  A_360_01_SQ5_A405_OPT_EKSKL : FbBinaryValue_Medium (2004) := (                _sDescription := 'Optimizer',                 _sActiveText := 'Utkoblet',                 _sInactiveText := 'Innkoblet'           );
  A_360_01_SQ5_A405_A1 : FbBinaryInput_Large (2008) := (                _sDescription := 'Luftmengde Sjeld',                 _sActiveText := 'Feil på luftmengde',                 _sInactiveText := 'Ingen feil',                 _udiNotificationClass := 22           );
  A_360_01_SQ5_A405_A2 : FbBinaryInput_Large (2009) := (                _sDescription := 'Kommunikasjonovervåking',                 _sActiveText := 'Kommunikasjonsfeil',                 _sInactiveText := 'Ingen feil',                 _udiNotificationClass := 22           );
  A_360_01_SQ4_A401_2_VOL : FbAnalogInput_Medium (2010) := (                _sDescription := 'Faktisk luftmengde',                 _rCov_Increment := 1,                 _eUnits := WagoTypesBacnet.eBACnetUnits.UNIT_CUBIC_METERS_PER_HOUR           );
  A_360_01_SQ4_A401_2_SP : FbAnalogValue_Medium (2015) := (                _sDescription := 'Settpunkt',                 _rCov_Increment := 1,                 _eUnits := WagoTypesBacnet.eBACnetUnits.UNIT_CUBIC_METERS_PER_HOUR           );
  A_360_01_SQ4_A401_2_VMIN : FbAnalogValue_Medium (2016) := (                _sDescription := 'Minste luftmengde',                 _rCov_Increment := 1,                 _eUnits := WagoTypesBacnet.eBACnetUnits.UNIT_CUBIC_METERS_PER_HOUR           );
  A_360_01_SQ4_A401_2_VMAX : FbAnalogValue_Medium (2017) := (                _sDescription := 'Største luftmengde',                 _rCov_Increment := 1,                 _eUnits := WagoTypesBacnet.eBACnetUnits.UNIT_CUBIC_METERS_PER_HOUR           );
  A_360_01_SQ4_A401_2_FB : FbAnalogInput_Medium (2011) := (                _sDescription := 'Spjeldvinkel',                 _rCov_Increment := 1,                 _eUnits := WagoTypesBacnet.eBACnetUnits.UNIT_PERCENT           );
  A_360_01_SQ4_A401_2_C : FbAnalogOutput_Medium (2005) := (                _sDescription := 'Pådrag',                 _rCov_Increment := 1,                 _eUnits := WagoTypesBacnet.eBACnetUnits.UNIT_PERCENT           );
  A_360_01_SQ4_A401_2_KMD : FbMultiStateValue_Large (2005) := (                _sDescription := 'Manuell overstyring',                 _udiNumberOfStates := 8           );
  A_360_01_SQ4_A401_2_OPT_EKSKL : FbBinaryValue_Medium (2005) := (                _sDescription := 'Optimizer',                 _sActiveText := 'Utkoblet',                 _sInactiveText := 'Innkoblet'           );
  A_360_01_SQ4_A401_2_A1 : FbBinaryInput_Large (2010) := (                _sDescription := 'Luftmengde Sjeld',                 _sActiveText := 'Feil på luftmengde',                 _sInactiveText := 'Ingen feil',                 _udiNotificationClass := 22           );
  A_360_01_SQ4_A401_2_A2 : FbBinaryInput_Large (2011) := (                _sDescription := 'Kommunikasjonovervåking',                 _sActiveText := 'Kommunikasjonsfeil',                 _sInactiveText := 'Ingen feil',                 _udiNotificationClass := 22           );
  A_360_01_SQ4_A401_1_VOL : FbAnalogInput_Medium (2012) := (                _sDescription := 'Faktisk luftmengde',                 _rCov_Increment := 1,                 _eUnits := WagoTypesBacnet.eBACnetUnits.UNIT_CUBIC_METERS_PER_HOUR           );
  A_360_01_SQ4_A401_1_SP : FbAnalogValue_Medium (2018) := (                _sDescription := 'Settpunkt',                 _rCov_Increment := 1,                 _eUnits := WagoTypesBacnet.eBACnetUnits.UNIT_CUBIC_METERS_PER_HOUR           );
  A_360_01_SQ4_A401_1_VMIN : FbAnalogValue_Medium (2019) := (                _sDescription := 'Minste luftmengde',                 _rCov_Increment := 1,                 _eUnits := WagoTypesBacnet.eBACnetUnits.UNIT_CUBIC_METERS_PER_HOUR           );
  A_360_01_SQ4_A401_1_VMAX : FbAnalogValue_Medium (2020) := (                _sDescription := 'Største luftmengde',                 _rCov_Increment := 1,                 _eUnits := WagoTypesBacnet.eBACnetUnits.UNIT_CUBIC_METERS_PER_HOUR           );
  A_360_01_SQ4_A401_1_FB : FbAnalogInput_Medium (2013) := (                _sDescription := 'Spjeldvinkel',                 _rCov_Increment := 1,                 _eUnits := WagoTypesBacnet.eBACnetUnits.UNIT_PERCENT           );
  A_360_01_SQ4_A401_1_C : FbAnalogOutput_Medium (2006) := (                _sDescription := 'Pådrag',                 _rCov_Increment := 1,                 _eUnits := WagoTypesBacnet.eBACnetUnits.UNIT_PERCENT           );
  A_360_01_SQ4_A401_1_KMD : FbMultiStateValue_Large (2006) := (                _sDescription := 'Manuell overstyring',                 _udiNumberOfStates := 8           );
  A_360_01_SQ4_A401_1_OPT_EKSKL : FbBinaryValue_Medium (2006) := (                _sDescription := 'Optimizer',                 _sActiveText := 'Utkoblet',                 _sInactiveText := 'Innkoblet'           );
  A_360_01_SQ4_A401_1_A1 : FbBinaryInput_Large (2012) := (                _sDescription := 'Luftmengde Sjeld',                 _sActiveText := 'Feil på luftmengde',                 _sInactiveText := 'Ingen feil',                 _udiNotificationClass := 22           );
  A_360_01_SQ4_A401_1_A2 : FbBinaryInput_Large (2013) := (                _sDescription := 'Kommunikasjonovervåking',                 _sActiveText := 'Kommunikasjonsfeil',                 _sInactiveText := 'Ingen feil',                 _udiNotificationClass := 22           );
  A_360_01_SQ4_A401_VOL : FbAnalogInput_Medium (2014) := (                _sDescription := 'Faktisk luftmengde',                 _rCov_Increment := 1,                 _eUnits := WagoTypesBacnet.eBACnetUnits.UNIT_CUBIC_METERS_PER_HOUR           );
  A_360_01_SQ4_A401_SP : FbAnalogValue_Medium (2021) := (                _sDescription := 'Settpunkt',                 _rCov_Increment := 1,                 _eUnits := WagoTypesBacnet.eBACnetUnits.UNIT_CUBIC_METERS_PER_HOUR           );
  A_360_01_SQ4_A401_VMIN : FbAnalogValue_Medium (2022) := (                _sDescription := 'Minste luftmengde',                 _rCov_Increment := 1,                 _eUnits := WagoTypesBacnet.eBACnetUnits.UNIT_CUBIC_METERS_PER_HOUR           );
  A_360_01_SQ4_A401_VMAX : FbAnalogValue_Medium (2023) := (                _sDescription := 'Største luftmengde',                 _rCov_Increment := 1,                 _eUnits := WagoTypesBacnet.eBACnetUnits.UNIT_CUBIC_METERS_PER_HOUR           );
  A_360_01_SQ4_A401_FB : FbAnalogInput_Medium (2015) := (                _sDescription := 'Spjeldvinkel',                 _rCov_Increment := 1,                 _eUnits := WagoTypesBacnet.eBACnetUnits.UNIT_PERCENT           );
  A_360_01_SQ4_A401_C : FbAnalogOutput_Medium (2007) := (                _sDescription := 'Pådrag',                 _rCov_Increment := 1,                 _eUnits := WagoTypesBacnet.eBACnetUnits.UNIT_PERCENT           );
  A_360_01_SQ4_A401_KMD : FbMultiStateValue_Large (2007) := (                _sDescription := 'Manuell overstyring',                 _udiNumberOfStates := 8           );
  A_360_01_SQ4_A401_OPT_EKSKL : FbBinaryValue_Medium (2007) := (                _sDescription := 'Optimizer',                 _sActiveText := 'Utkoblet',                 _sInactiveText := 'Innkoblet'           );
  A_360_01_SQ4_A401_A1 : FbBinaryInput_Large (2014) := (                _sDescription := 'Luftmengde Sjeld',                 _sActiveText := 'Feil på luftmengde',                 _sInactiveText := 'Ingen feil',                 _udiNotificationClass := 22           );
  A_360_01_SQ4_A401_A2 : FbBinaryInput_Large (2015) := (                _sDescription := 'Kommunikasjonovervåking',                 _sActiveText := 'Kommunikasjonsfeil',                 _sInactiveText := 'Ingen feil',                 _udiNotificationClass := 22           );
  A_360_01_SQ4_A406_VOL : FbAnalogInput_Medium (2016) := (                _sDescription := 'Faktisk luftmengde',                 _rCov_Increment := 1,                 _eUnits := WagoTypesBacnet.eBACnetUnits.UNIT_CUBIC_METERS_PER_HOUR           );
  A_360_01_SQ4_A406_SP : FbAnalogValue_Medium (2024) := (                _sDescription := 'Settpunkt',                 _rCov_Increment := 1,                 _eUnits := WagoTypesBacnet.eBACnetUnits.UNIT_CUBIC_METERS_PER_HOUR           );
  A_360_01_SQ4_A406_VMIN : FbAnalogValue_Medium (2025) := (                _sDescription := 'Minste luftmengde',                 _rCov_Increment := 1,                 _eUnits := WagoTypesBacnet.eBACnetUnits.UNIT_CUBIC_METERS_PER_HOUR           );
  A_360_01_SQ4_A406_VMAX : FbAnalogValue_Medium (2026) := (                _sDescription := 'Største luftmengde',                 _rCov_Increment := 1,                 _eUnits := WagoTypesBacnet.eBACnetUnits.UNIT_CUBIC_METERS_PER_HOUR           );
  A_360_01_SQ4_A406_FB : FbAnalogInput_Medium (2017) := (                _sDescription := 'Spjeldvinkel',                 _rCov_Increment := 1,                 _eUnits := WagoTypesBacnet.eBACnetUnits.UNIT_PERCENT           );
  A_360_01_SQ4_A406_C : FbAnalogOutput_Medium (2008) := (                _sDescription := 'Pådrag',                 _rCov_Increment := 1,                 _eUnits := WagoTypesBacnet.eBACnetUnits.UNIT_PERCENT           );
  A_360_01_SQ4_A406_KMD : FbMultiStateValue_Large (2008) := (                _sDescription := 'Manuell overstyring',                 _udiNumberOfStates := 8           );
  A_360_01_SQ4_A406_OPT_EKSKL : FbBinaryValue_Medium (2008) := (                _sDescription := 'Optimizer',                 _sActiveText := 'Utkoblet',                 _sInactiveText := 'Innkoblet'           );
  A_360_01_SQ4_A406_A1 : FbBinaryInput_Large (2016) := (                _sDescription := 'Luftmengde Sjeld',                 _sActiveText := 'Feil på luftmengde',                 _sInactiveText := 'Ingen feil',                 _udiNotificationClass := 22           );
  A_360_01_SQ4_A406_A2 : FbBinaryInput_Large (2017) := (                _sDescription := 'Kommunikasjonovervåking',                 _sActiveText := 'Kommunikasjonsfeil',                 _sInactiveText := 'Ingen feil',                 _udiNotificationClass := 22           );
  A_360_01_SQ4_A408_VOL : FbAnalogInput_Medium (2018) := (                _sDescription := 'Faktisk luftmengde',                 _rCov_Increment := 1,                 _eUnits := WagoTypesBacnet.eBACnetUnits.UNIT_CUBIC_METERS_PER_HOUR           );
  A_360_01_SQ4_A408_SP : FbAnalogValue_Medium (2027) := (                _sDescription := 'Settpunkt',                 _rCov_Increment := 1,                 _eUnits := WagoTypesBacnet.eBACnetUnits.UNIT_CUBIC_METERS_PER_HOUR           );
  A_360_01_SQ4_A408_VMIN : FbAnalogValue_Medium (2028) := (                _sDescription := 'Minste luftmengde',                 _rCov_Increment := 1,                 _eUnits := WagoTypesBacnet.eBACnetUnits.UNIT_CUBIC_METERS_PER_HOUR           );
  A_360_01_SQ4_A408_VMAX : FbAnalogValue_Medium (2029) := (                _sDescription := 'Største luftmengde',                 _rCov_Increment := 1,                 _eUnits := WagoTypesBacnet.eBACnetUnits.UNIT_CUBIC_METERS_PER_HOUR           );
  A_360_01_SQ4_A408_FB : FbAnalogInput_Medium (2019) := (                _sDescription := 'Spjeldvinkel',                 _rCov_Increment := 1,                 _eUnits := WagoTypesBacnet.eBACnetUnits.UNIT_PERCENT           );
  A_360_01_SQ4_A408_C : FbAnalogOutput_Medium (2009) := (                _sDescription := 'Pådrag',                 _rCov_Increment := 1,                 _eUnits := WagoTypesBacnet.eBACnetUnits.UNIT_PERCENT           );
  A_360_01_SQ4_A408_KMD : FbMultiStateValue_Large (2009) := (                _sDescription := 'Manuell overstyring',                 _udiNumberOfStates := 8           );
  A_360_01_SQ4_A408_OPT_EKSKL : FbBinaryValue_Medium (2009) := (                _sDescription := 'Optimizer',                 _sActiveText := 'Utkoblet',                 _sInactiveText := 'Innkoblet'           );
  A_360_01_SQ4_A408_A1 : FbBinaryInput_Large (2018) := (                _sDescription := 'Luftmengde Sjeld',                 _sActiveText := 'Feil på luftmengde',                 _sInactiveText := 'Ingen feil',                 _udiNotificationClass := 22           );
  A_360_01_SQ4_A408_A2 : FbBinaryInput_Large (2019) := (                _sDescription := 'Kommunikasjonovervåking',                 _sActiveText := 'Kommunikasjonsfeil',                 _sInactiveText := 'Ingen feil',                 _udiNotificationClass := 22           );
  A_360_01_SQ4_A410_1_VOL : FbAnalogInput_Medium (2020) := (                _sDescription := 'Faktisk luftmengde',                 _rCov_Increment := 1,                 _eUnits := WagoTypesBacnet.eBACnetUnits.UNIT_CUBIC_METERS_PER_HOUR           );
  A_360_01_SQ4_A410_1_SP : FbAnalogValue_Medium (2030) := (                _sDescription := 'Settpunkt',                 _rCov_Increment := 1,                 _eUnits := WagoTypesBacnet.eBACnetUnits.UNIT_CUBIC_METERS_PER_HOUR           );
  A_360_01_SQ4_A410_1_VMIN : FbAnalogValue_Medium (2031) := (                _sDescription := 'Minste luftmengde',                 _rCov_Increment := 1,                 _eUnits := WagoTypesBacnet.eBACnetUnits.UNIT_CUBIC_METERS_PER_HOUR           );
  A_360_01_SQ4_A410_1_VMAX : FbAnalogValue_Medium (2032) := (                _sDescription := 'Største luftmengde',                 _rCov_Increment := 1,                 _eUnits := WagoTypesBacnet.eBACnetUnits.UNIT_CUBIC_METERS_PER_HOUR           );
  A_360_01_SQ4_A410_1_FB : FbAnalogInput_Medium (2021) := (                _sDescription := 'Spjeldvinkel',                 _rCov_Increment := 1,                 _eUnits := WagoTypesBacnet.eBACnetUnits.UNIT_PERCENT           );
  A_360_01_SQ4_A410_1_C : FbAnalogOutput_Medium (2010) := (                _sDescription := 'Pådrag',                 _rCov_Increment := 1,                 _eUnits := WagoTypesBacnet.eBACnetUnits.UNIT_PERCENT           );
  A_360_01_SQ4_A410_1_KMD : FbMultiStateValue_Large (2010) := (                _sDescription := 'Manuell overstyring',                 _udiNumberOfStates := 8           );
  A_360_01_SQ4_A410_1_OPT_EKSKL : FbBinaryValue_Medium (2010) := (                _sDescription := 'Optimizer',                 _sActiveText := 'Utkoblet',                 _sInactiveText := 'Innkoblet'           );
  A_360_01_SQ4_A410_1_A1 : FbBinaryInput_Large (2020) := (                _sDescription := 'Luftmengde Sjeld',                 _sActiveText := 'Feil på luftmengde',                 _sInactiveText := 'Ingen feil',                 _udiNotificationClass := 22           );
  A_360_01_SQ4_A410_1_A2 : FbBinaryInput_Large (2021) := (                _sDescription := 'Kommunikasjonovervåking',                 _sActiveText := 'Kommunikasjonsfeil',                 _sInactiveText := 'Ingen feil',                 _udiNotificationClass := 22           );
  A_360_01_SQ4_A410_2_VOL : FbAnalogInput_Medium (2022) := (                _sDescription := 'Faktisk luftmengde',                 _rCov_Increment := 1,                 _eUnits := WagoTypesBacnet.eBACnetUnits.UNIT_CUBIC_METERS_PER_HOUR           );
  A_360_01_SQ4_A410_2_SP : FbAnalogValue_Medium (2033) := (                _sDescription := 'Settpunkt',                 _rCov_Increment := 1,                 _eUnits := WagoTypesBacnet.eBACnetUnits.UNIT_CUBIC_METERS_PER_HOUR           );
  A_360_01_SQ4_A410_2_VMIN : FbAnalogValue_Medium (2034) := (                _sDescription := 'Minste luftmengde',                 _rCov_Increment := 1,                 _eUnits := WagoTypesBacnet.eBACnetUnits.UNIT_CUBIC_METERS_PER_HOUR           );
  A_360_01_SQ4_A410_2_VMAX : FbAnalogValue_Medium (2035) := (                _sDescription := 'Største luftmengde',                 _rCov_Increment := 1,                 _eUnits := WagoTypesBacnet.eBACnetUnits.UNIT_CUBIC_METERS_PER_HOUR           );
  A_360_01_SQ4_A410_2_FB : FbAnalogInput_Medium (2023) := (                _sDescription := 'Spjeldvinkel',                 _rCov_Increment := 1,                 _eUnits := WagoTypesBacnet.eBACnetUnits.UNIT_PERCENT           );
  A_360_01_SQ4_A410_2_C : FbAnalogOutput_Medium (2011) := (                _sDescription := 'Pådrag',                 _rCov_Increment := 1,                 _eUnits := WagoTypesBacnet.eBACnetUnits.UNIT_PERCENT           );
  A_360_01_SQ4_A410_2_KMD : FbMultiStateValue_Large (2011) := (                _sDescription := 'Manuell overstyring',                 _udiNumberOfStates := 8           );
  A_360_01_SQ4_A410_2_OPT_EKSKL : FbBinaryValue_Medium (2011) := (                _sDescription := 'Optimizer',                 _sActiveText := 'Utkoblet',                 _sInactiveText := 'Innkoblet'           );
  A_360_01_SQ4_A410_2_A1 : FbBinaryInput_Large (2022) := (                _sDescription := 'Luftmengde Sjeld',                 _sActiveText := 'Feil på luftmengde',                 _sInactiveText := 'Ingen feil',                 _udiNotificationClass := 22           );
  A_360_01_SQ4_A410_2_A2 : FbBinaryInput_Large (2023) := (                _sDescription := 'Kommunikasjonovervåking',                 _sActiveText := 'Kommunikasjonsfeil',                 _sInactiveText := 'Ingen feil',                 _udiNotificationClass := 22           );
  A_360_01_SQ4_A410_3_VOL : FbAnalogInput_Medium (2024) := (                _sDescription := 'Faktisk luftmengde',                 _rCov_Increment := 1,                 _eUnits := WagoTypesBacnet.eBACnetUnits.UNIT_CUBIC_METERS_PER_HOUR           );
  A_360_01_SQ4_A410_3_SP : FbAnalogValue_Medium (2036) := (                _sDescription := 'Settpunkt',                 _rCov_Increment := 1,                 _eUnits := WagoTypesBacnet.eBACnetUnits.UNIT_CUBIC_METERS_PER_HOUR           );
  A_360_01_SQ4_A410_3_VMIN : FbAnalogValue_Medium (2037) := (                _sDescription := 'Minste luftmengde',                 _rCov_Increment := 1,                 _eUnits := WagoTypesBacnet.eBACnetUnits.UNIT_CUBIC_METERS_PER_HOUR           );
  A_360_01_SQ4_A410_3_VMAX : FbAnalogValue_Medium (2038) := (                _sDescription := 'Største luftmengde',                 _rCov_Increment := 1,                 _eUnits := WagoTypesBacnet.eBACnetUnits.UNIT_CUBIC_METERS_PER_HOUR           );
  A_360_01_SQ4_A410_3_FB : FbAnalogInput_Medium (2025) := (                _sDescription := 'Spjeldvinkel',                 _rCov_Increment := 1,                 _eUnits := WagoTypesBacnet.eBACnetUnits.UNIT_PERCENT           );
  A_360_01_SQ4_A410_3_C : FbAnalogOutput_Medium (2012) := (                _sDescription := 'Pådrag',                 _rCov_Increment := 1,                 _eUnits := WagoTypesBacnet.eBACnetUnits.UNIT_PERCENT           );
  A_360_01_SQ4_A410_3_KMD : FbMultiStateValue_Large (2012) := (                _sDescription := 'Manuell overstyring',                 _udiNumberOfStates := 8           );
  A_360_01_SQ4_A410_3_OPT_EKSKL : FbBinaryValue_Medium (2012) := (                _sDescription := 'Optimizer',                 _sActiveText := 'Utkoblet',                 _sInactiveText := 'Innkoblet'           );
  A_360_01_SQ4_A410_3_A1 : FbBinaryInput_Large (2024) := (                _sDescription := 'Luftmengde Sjeld',                 _sActiveText := 'Feil på luftmengde',                 _sInactiveText := 'Ingen feil',                 _udiNotificationClass := 22           );
  A_360_01_SQ4_A410_3_A2 : FbBinaryInput_Large (2025) := (                _sDescription := 'Kommunikasjonovervåking',                 _sActiveText := 'Kommunikasjonsfeil',                 _sInactiveText := 'Ingen feil',                 _udiNotificationClass := 22           );
  A_360_01_SQ4_A410_4_VOL : FbAnalogInput_Medium (2026) := (                _sDescription := 'Faktisk luftmengde',                 _rCov_Increment := 1,                 _eUnits := WagoTypesBacnet.eBACnetUnits.UNIT_CUBIC_METERS_PER_HOUR           );
  A_360_01_SQ4_A410_4_SP : FbAnalogValue_Medium (2039) := (                _sDescription := 'Settpunkt',                 _rCov_Increment := 1,                 _eUnits := WagoTypesBacnet.eBACnetUnits.UNIT_CUBIC_METERS_PER_HOUR           );
  A_360_01_SQ4_A410_4_VMIN : FbAnalogValue_Medium (2040) := (                _sDescription := 'Minste luftmengde',                 _rCov_Increment := 1,                 _eUnits := WagoTypesBacnet.eBACnetUnits.UNIT_CUBIC_METERS_PER_HOUR           );
  A_360_01_SQ4_A410_4_VMAX : FbAnalogValue_Medium (2041) := (                _sDescription := 'Største luftmengde',                 _rCov_Increment := 1,                 _eUnits := WagoTypesBacnet.eBACnetUnits.UNIT_CUBIC_METERS_PER_HOUR           );
  A_360_01_SQ4_A410_4_FB : FbAnalogInput_Medium (2027) := (                _sDescription := 'Spjeldvinkel',                 _rCov_Increment := 1,                 _eUnits := WagoTypesBacnet.eBACnetUnits.UNIT_PERCENT           );
  A_360_01_SQ4_A410_4_C : FbAnalogOutput_Medium (2013) := (                _sDescription := 'Pådrag',                 _rCov_Increment := 1,                 _eUnits := WagoTypesBacnet.eBACnetUnits.UNIT_PERCENT           );
  A_360_01_SQ4_A410_4_KMD : FbMultiStateValue_Large (2013) := (                _sDescription := 'Manuell overstyring',                 _udiNumberOfStates := 8           );
  A_360_01_SQ4_A410_4_OPT_EKSKL : FbBinaryValue_Medium (2013) := (                _sDescription := 'Optimizer',                 _sActiveText := 'Utkoblet',                 _sInactiveText := 'Innkoblet'           );
  A_360_01_SQ4_A410_4_A1 : FbBinaryInput_Large (2026) := (                _sDescription := 'Luftmengde Sjeld',                 _sActiveText := 'Feil på luftmengde',                 _sInactiveText := 'Ingen feil',                 _udiNotificationClass := 22           );
  A_360_01_SQ4_A410_4_A2 : FbBinaryInput_Large (2027) := (                _sDescription := 'Kommunikasjonovervåking',                 _sActiveText := 'Kommunikasjonsfeil',                 _sInactiveText := 'Ingen feil',                 _udiNotificationClass := 22           );
  A_360_01_SQ4_A410_5_VOL : FbAnalogInput_Medium (2028) := (                _sDescription := 'Faktisk luftmengde',                 _rCov_Increment := 1,                 _eUnits := WagoTypesBacnet.eBACnetUnits.UNIT_CUBIC_METERS_PER_HOUR           );
  A_360_01_SQ4_A410_5_SP : FbAnalogValue_Medium (2042) := (                _sDescription := 'Settpunkt',                 _rCov_Increment := 1,                 _eUnits := WagoTypesBacnet.eBACnetUnits.UNIT_CUBIC_METERS_PER_HOUR           );
  A_360_01_SQ4_A410_5_VMIN : FbAnalogValue_Medium (2043) := (                _sDescription := 'Minste luftmengde',                 _rCov_Increment := 1,                 _eUnits := WagoTypesBacnet.eBACnetUnits.UNIT_CUBIC_METERS_PER_HOUR           );
  A_360_01_SQ4_A410_5_VMAX : FbAnalogValue_Medium (2044) := (                _sDescription := 'Største luftmengde',                 _rCov_Increment := 1,                 _eUnits := WagoTypesBacnet.eBACnetUnits.UNIT_CUBIC_METERS_PER_HOUR           );
  A_360_01_SQ4_A410_5_FB : FbAnalogInput_Medium (2029) := (                _sDescription := 'Spjeldvinkel',                 _rCov_Increment := 1,                 _eUnits := WagoTypesBacnet.eBACnetUnits.UNIT_PERCENT           );
  A_360_01_SQ4_A410_5_C : FbAnalogOutput_Medium (2014) := (                _sDescription := 'Pådrag',                 _rCov_Increment := 1,                 _eUnits := WagoTypesBacnet.eBACnetUnits.UNIT_PERCENT           );
  A_360_01_SQ4_A410_5_KMD : FbMultiStateValue_Large (2014) := (                _sDescription := 'Manuell overstyring',                 _udiNumberOfStates := 8           );
  A_360_01_SQ4_A410_5_OPT_EKSKL : FbBinaryValue_Medium (2014) := (                _sDescription := 'Optimizer',                 _sActiveText := 'Utkoblet',                 _sInactiveText := 'Innkoblet'           );
  A_360_01_SQ4_A410_5_A1 : FbBinaryInput_Large (2028) := (                _sDescription := 'Luftmengde Sjeld',                 _sActiveText := 'Feil på luftmengde',                 _sInactiveText := 'Ingen feil',                 _udiNotificationClass := 22           );
  A_360_01_SQ4_A410_5_A2 : FbBinaryInput_Large (2029) := (                _sDescription := 'Kommunikasjonovervåking',                 _sActiveText := 'Kommunikasjonsfeil',                 _sInactiveText := 'Ingen feil',                 _udiNotificationClass := 22           );
  A_360_01_SQ4_A412_VOL : FbAnalogInput_Medium (2030) := (                _sDescription := 'Faktisk luftmengde',                 _rCov_Increment := 1,                 _eUnits := WagoTypesBacnet.eBACnetUnits.UNIT_CUBIC_METERS_PER_HOUR           );
  A_360_01_SQ4_A412_SP : FbAnalogValue_Medium (2045) := (                _sDescription := 'Settpunkt',                 _rCov_Increment := 1,                 _eUnits := WagoTypesBacnet.eBACnetUnits.UNIT_CUBIC_METERS_PER_HOUR           );
  A_360_01_SQ4_A412_VMIN : FbAnalogValue_Medium (2046) := (                _sDescription := 'Minste luftmengde',                 _rCov_Increment := 1,                 _eUnits := WagoTypesBacnet.eBACnetUnits.UNIT_CUBIC_METERS_PER_HOUR           );
  A_360_01_SQ4_A412_VMAX : FbAnalogValue_Medium (2047) := (                _sDescription := 'Største luftmengde',                 _rCov_Increment := 1,                 _eUnits := WagoTypesBacnet.eBACnetUnits.UNIT_CUBIC_METERS_PER_HOUR           );
  A_360_01_SQ4_A412_FB : FbAnalogInput_Medium (2031) := (                _sDescription := 'Spjeldvinkel',                 _rCov_Increment := 1,                 _eUnits := WagoTypesBacnet.eBACnetUnits.UNIT_PERCENT           );
  A_360_01_SQ4_A412_C : FbAnalogOutput_Medium (2015) := (                _sDescription := 'Pådrag',                 _rCov_Increment := 1,                 _eUnits := WagoTypesBacnet.eBACnetUnits.UNIT_PERCENT           );
  A_360_01_SQ4_A412_KMD : FbMultiStateValue_Large (2015) := (                _sDescription := 'Manuell overstyring',                 _udiNumberOfStates := 8           );
  A_360_01_SQ4_A412_OPT_EKSKL : FbBinaryValue_Medium (2015) := (                _sDescription := 'Optimizer',                 _sActiveText := 'Utkoblet',                 _sInactiveText := 'Innkoblet'           );
  A_360_01_SQ4_A412_A1 : FbBinaryInput_Large (2030) := (                _sDescription := 'Luftmengde Sjeld',                 _sActiveText := 'Feil på luftmengde',                 _sInactiveText := 'Ingen feil',                 _udiNotificationClass := 22           );
  A_360_01_SQ4_A412_A2 : FbBinaryInput_Large (2031) := (                _sDescription := 'Kommunikasjonovervåking',                 _sActiveText := 'Kommunikasjonsfeil',                 _sInactiveText := 'Ingen feil',                 _udiNotificationClass := 22           );
  A_360_01_SQ4_A413_VOL : FbAnalogInput_Medium (2032) := (                _sDescription := 'Faktisk luftmengde',                 _rCov_Increment := 1,                 _eUnits := WagoTypesBacnet.eBACnetUnits.UNIT_CUBIC_METERS_PER_HOUR           );
  A_360_01_SQ4_A413_SP : FbAnalogValue_Medium (2048) := (                _sDescription := 'Settpunkt',                 _rCov_Increment := 1,                 _eUnits := WagoTypesBacnet.eBACnetUnits.UNIT_CUBIC_METERS_PER_HOUR           );
  A_360_01_SQ4_A413_VMIN : FbAnalogValue_Medium (2049) := (                _sDescription := 'Minste luftmengde',                 _rCov_Increment := 1,                 _eUnits := WagoTypesBacnet.eBACnetUnits.UNIT_CUBIC_METERS_PER_HOUR           );
  A_360_01_SQ4_A413_VMAX : FbAnalogValue_Medium (2050) := (                _sDescription := 'Største luftmengde',                 _rCov_Increment := 1,                 _eUnits := WagoTypesBacnet.eBACnetUnits.UNIT_CUBIC_METERS_PER_HOUR           );
  A_360_01_SQ4_A413_FB : FbAnalogInput_Medium (2033) := (                _sDescription := 'Spjeldvinkel',                 _rCov_Increment := 1,                 _eUnits := WagoTypesBacnet.eBACnetUnits.UNIT_PERCENT           );
  A_360_01_SQ4_A413_C : FbAnalogOutput_Medium (2016) := (                _sDescription := 'Pådrag',                 _rCov_Increment := 1,                 _eUnits := WagoTypesBacnet.eBACnetUnits.UNIT_PERCENT           );
  A_360_01_SQ4_A413_KMD : FbMultiStateValue_Large (2016) := (                _sDescription := 'Manuell overstyring',                 _udiNumberOfStates := 8           );
  A_360_01_SQ4_A413_OPT_EKSKL : FbBinaryValue_Medium (2016) := (                _sDescription := 'Optimizer',                 _sActiveText := 'Utkoblet',                 _sInactiveText := 'Innkoblet'           );
  A_360_01_SQ4_A413_A1 : FbBinaryInput_Large (2032) := (                _sDescription := 'Luftmengde Sjeld',                 _sActiveText := 'Feil på luftmengde',                 _sInactiveText := 'Ingen feil',                 _udiNotificationClass := 22           );
  A_360_01_SQ4_A413_A2 : FbBinaryInput_Large (2033) := (                _sDescription := 'Kommunikasjonovervåking',                 _sActiveText := 'Kommunikasjonsfeil',                 _sInactiveText := 'Ingen feil',                 _udiNotificationClass := 22           );
  A_360_01_SK4_A415_VOL : FbAnalogInput_Medium (2034) := (                _sDescription := 'Faktisk luftmengde',                 _rCov_Increment := 1,                 _eUnits := WagoTypesBacnet.eBACnetUnits.UNIT_CUBIC_METERS_PER_HOUR           );
  A_360_01_SK4_A415_SP : FbAnalogValue_Medium (2051) := (                _sDescription := 'Settpunkt',                 _rCov_Increment := 1,                 _eUnits := WagoTypesBacnet.eBACnetUnits.UNIT_CUBIC_METERS_PER_HOUR           );
  A_360_01_SK4_A415_VMIN : FbAnalogValue_Medium (2052) := (                _sDescription := 'Minste luftmengde',                 _rCov_Increment := 1,                 _eUnits := WagoTypesBacnet.eBACnetUnits.UNIT_CUBIC_METERS_PER_HOUR           );
  A_360_01_SK4_A415_VMAX : FbAnalogValue_Medium (2053) := (                _sDescription := 'Største luftmengde',                 _rCov_Increment := 1,                 _eUnits := WagoTypesBacnet.eBACnetUnits.UNIT_CUBIC_METERS_PER_HOUR           );
  A_360_01_SK4_A415_FB : FbAnalogInput_Medium (2035) := (                _sDescription := 'Spjeldvinkel',                 _rCov_Increment := 1,                 _eUnits := WagoTypesBacnet.eBACnetUnits.UNIT_PERCENT           );
  A_360_01_SK4_A415_C : FbAnalogOutput_Medium (2017) := (                _sDescription := 'Pådrag',                 _rCov_Increment := 1,                 _eUnits := WagoTypesBacnet.eBACnetUnits.UNIT_PERCENT           );
  A_360_01_SK4_A415_KMD : FbMultiStateValue_Large (2017) := (                _sDescription := 'Manuell overstyring',                 _udiNumberOfStates := 8           );
  A_360_01_SK4_A415_OPT_EKSKL : FbBinaryValue_Medium (2017) := (                _sDescription := 'Optimizer',                 _sActiveText := 'Utkoblet',                 _sInactiveText := 'Innkoblet'           );
  A_360_01_SK4_A415_A1 : FbBinaryInput_Large (2034) := (                _sDescription := 'Luftmengde Sjeld',                 _sActiveText := 'Feil på luftmengde',                 _sInactiveText := 'Ingen feil',                 _udiNotificationClass := 22           );
  A_360_01_SK4_A415_A2 : FbBinaryInput_Large (2035) := (                _sDescription := 'Kommunikasjonovervåking',                 _sActiveText := 'Kommunikasjonsfeil',                 _sInactiveText := 'Ingen feil',                 _udiNotificationClass := 22           );
  A_360_01_SK5_A415_VOL : FbAnalogInput_Medium (2036) := (                _sDescription := 'Faktisk luftmengde',                 _rCov_Increment := 1,                 _eUnits := WagoTypesBacnet.eBACnetUnits.UNIT_CUBIC_METERS_PER_HOUR           );
  A_360_01_SK5_A415_SP : FbAnalogValue_Medium (2054) := (                _sDescription := 'Settpunkt',                 _rCov_Increment := 1,                 _eUnits := WagoTypesBacnet.eBACnetUnits.UNIT_CUBIC_METERS_PER_HOUR           );
  A_360_01_SK5_A415_VMIN : FbAnalogValue_Medium (2055) := (                _sDescription := 'Minste luftmengde',                 _rCov_Increment := 1,                 _eUnits := WagoTypesBacnet.eBACnetUnits.UNIT_CUBIC_METERS_PER_HOUR           );
  A_360_01_SK5_A415_VMAX : FbAnalogValue_Medium (2056) := (                _sDescription := 'Største luftmengde',                 _rCov_Increment := 1,                 _eUnits := WagoTypesBacnet.eBACnetUnits.UNIT_CUBIC_METERS_PER_HOUR           );
  A_360_01_SK5_A415_FB : FbAnalogInput_Medium (2037) := (                _sDescription := 'Spjeldvinkel',                 _rCov_Increment := 1,                 _eUnits := WagoTypesBacnet.eBACnetUnits.UNIT_PERCENT           );
  A_360_01_SK5_A415_C : FbAnalogOutput_Medium (2018) := (                _sDescription := 'Pådrag',                 _rCov_Increment := 1,                 _eUnits := WagoTypesBacnet.eBACnetUnits.UNIT_PERCENT           );
  A_360_01_SK5_A415_KMD : FbMultiStateValue_Large (2018) := (                _sDescription := 'Manuell overstyring',                 _udiNumberOfStates := 8           );
  A_360_01_SK5_A415_OPT_EKSKL : FbBinaryValue_Medium (2018) := (                _sDescription := 'Optimizer',                 _sActiveText := 'Utkoblet',                 _sInactiveText := 'Innkoblet'           );
  A_360_01_SK5_A415_A1 : FbBinaryInput_Large (2036) := (                _sDescription := 'Luftmengde Sjeld',                 _sActiveText := 'Feil på luftmengde',                 _sInactiveText := 'Ingen feil',                 _udiNotificationClass := 22           );
  A_360_01_SK5_A415_A2 : FbBinaryInput_Large (2037) := (                _sDescription := 'Kommunikasjonovervåking',                 _sActiveText := 'Kommunikasjonsfeil',                 _sInactiveText := 'Ingen feil',                 _udiNotificationClass := 22           );
  A_360_01_SK5_A418_VOL : FbAnalogInput_Medium (2038) := (                _sDescription := 'Faktisk luftmengde',                 _rCov_Increment := 1,                 _eUnits := WagoTypesBacnet.eBACnetUnits.UNIT_CUBIC_METERS_PER_HOUR           );
  A_360_01_SK5_A418_SP : FbAnalogValue_Medium (2057) := (                _sDescription := 'Settpunkt',                 _rCov_Increment := 1,                 _eUnits := WagoTypesBacnet.eBACnetUnits.UNIT_CUBIC_METERS_PER_HOUR           );
  A_360_01_SK5_A418_VMIN : FbAnalogValue_Medium (2058) := (                _sDescription := 'Minste luftmengde',                 _rCov_Increment := 1,                 _eUnits := WagoTypesBacnet.eBACnetUnits.UNIT_CUBIC_METERS_PER_HOUR           );
  A_360_01_SK5_A418_VMAX : FbAnalogValue_Medium (2059) := (                _sDescription := 'Største luftmengde',                 _rCov_Increment := 1,                 _eUnits := WagoTypesBacnet.eBACnetUnits.UNIT_CUBIC_METERS_PER_HOUR           );
  A_360_01_SK5_A418_FB : FbAnalogInput_Medium (2039) := (                _sDescription := 'Spjeldvinkel',                 _rCov_Increment := 1,                 _eUnits := WagoTypesBacnet.eBACnetUnits.UNIT_PERCENT           );
  A_360_01_SK5_A418_C : FbAnalogOutput_Medium (2019) := (                _sDescription := 'Pådrag',                 _rCov_Increment := 1,                 _eUnits := WagoTypesBacnet.eBACnetUnits.UNIT_PERCENT           );
  A_360_01_SK5_A418_KMD : FbMultiStateValue_Large (2019) := (                _sDescription := 'Manuell overstyring',                 _udiNumberOfStates := 8           );
  A_360_01_SK5_A418_OPT_EKSKL : FbBinaryValue_Medium (2019) := (                _sDescription := 'Optimizer',                 _sActiveText := 'Utkoblet',                 _sInactiveText := 'Innkoblet'           );
  A_360_01_SK5_A418_A1 : FbBinaryInput_Large (2038) := (                _sDescription := 'Luftmengde Sjeld',                 _sActiveText := 'Feil på luftmengde',                 _sInactiveText := 'Ingen feil',                 _udiNotificationClass := 22           );
  A_360_01_SK5_A418_A2 : FbBinaryInput_Large (2039) := (                _sDescription := 'Kommunikasjonovervåking',                 _sActiveText := 'Kommunikasjonsfeil',                 _sInactiveText := 'Ingen feil',                 _udiNotificationClass := 22           );
  A_360_01_SK4_A417_VOL : FbAnalogInput_Medium (2040) := (                _sDescription := 'Faktisk luftmengde',                 _rCov_Increment := 1,                 _eUnits := WagoTypesBacnet.eBACnetUnits.UNIT_CUBIC_METERS_PER_HOUR           );
  A_360_01_SK4_A417_SP : FbAnalogValue_Medium (2060) := (                _sDescription := 'Settpunkt',                 _rCov_Increment := 1,                 _eUnits := WagoTypesBacnet.eBACnetUnits.UNIT_CUBIC_METERS_PER_HOUR           );
  A_360_01_SK4_A417_VMIN : FbAnalogValue_Medium (2061) := (                _sDescription := 'Minste luftmengde',                 _rCov_Increment := 1,                 _eUnits := WagoTypesBacnet.eBACnetUnits.UNIT_CUBIC_METERS_PER_HOUR           );
  A_360_01_SK4_A417_VMAX : FbAnalogValue_Medium (2062) := (                _sDescription := 'Største luftmengde',                 _rCov_Increment := 1,                 _eUnits := WagoTypesBacnet.eBACnetUnits.UNIT_CUBIC_METERS_PER_HOUR           );
  A_360_01_SK4_A417_FB : FbAnalogInput_Medium (2041) := (                _sDescription := 'Spjeldvinkel',                 _rCov_Increment := 1,                 _eUnits := WagoTypesBacnet.eBACnetUnits.UNIT_PERCENT           );
  A_360_01_SK4_A417_C : FbAnalogOutput_Medium (2020) := (                _sDescription := 'Pådrag',                 _rCov_Increment := 1,                 _eUnits := WagoTypesBacnet.eBACnetUnits.UNIT_PERCENT           );
  A_360_01_SK4_A417_KMD : FbMultiStateValue_Large (2020) := (                _sDescription := 'Manuell overstyring',                 _udiNumberOfStates := 8           );
  A_360_01_SK4_A417_OPT_EKSKL : FbBinaryValue_Medium (2020) := (                _sDescription := 'Optimizer',                 _sActiveText := 'Utkoblet',                 _sInactiveText := 'Innkoblet'           );
  A_360_01_SK4_A417_A1 : FbBinaryInput_Large (2040) := (                _sDescription := 'Luftmengde Sjeld',                 _sActiveText := 'Feil på luftmengde',                 _sInactiveText := 'Ingen feil',                 _udiNotificationClass := 22           );
  A_360_01_SK4_A417_A2 : FbBinaryInput_Large (2041) := (                _sDescription := 'Kommunikasjonovervåking',                 _sActiveText := 'Kommunikasjonsfeil',                 _sInactiveText := 'Ingen feil',                 _udiNotificationClass := 22           );
  A_360_01_SQ5_C411_VOL : FbAnalogInput_Medium (2042) := (                _sDescription := 'Faktisk luftmengde',                 _rCov_Increment := 1,                 _eUnits := WagoTypesBacnet.eBACnetUnits.UNIT_CUBIC_METERS_PER_HOUR           );
  A_360_01_SQ5_C411_SP : FbAnalogValue_Medium (2063) := (                _sDescription := 'Settpunkt',                 _rCov_Increment := 1,                 _eUnits := WagoTypesBacnet.eBACnetUnits.UNIT_CUBIC_METERS_PER_HOUR           );
  A_360_01_SQ5_C411_VMIN : FbAnalogValue_Medium (2064) := (                _sDescription := 'Minste luftmengde',                 _rCov_Increment := 1,                 _eUnits := WagoTypesBacnet.eBACnetUnits.UNIT_CUBIC_METERS_PER_HOUR           );
  A_360_01_SQ5_C411_VMAX : FbAnalogValue_Medium (2065) := (                _sDescription := 'Største luftmengde',                 _rCov_Increment := 1,                 _eUnits := WagoTypesBacnet.eBACnetUnits.UNIT_CUBIC_METERS_PER_HOUR           );
  A_360_01_SQ5_C411_FB : FbAnalogInput_Medium (2043) := (                _sDescription := 'Spjeldvinkel',                 _rCov_Increment := 1,                 _eUnits := WagoTypesBacnet.eBACnetUnits.UNIT_PERCENT           );
  A_360_01_SQ5_C411_C : FbAnalogOutput_Medium (2021) := (                _sDescription := 'Pådrag',                 _rCov_Increment := 1,                 _eUnits := WagoTypesBacnet.eBACnetUnits.UNIT_PERCENT           );
  A_360_01_SQ5_C411_KMD : FbMultiStateValue_Large (2021) := (                _sDescription := 'Manuell overstyring',                 _udiNumberOfStates := 8           );
  A_360_01_SQ5_C411_OPT_EKSKL : FbBinaryValue_Medium (2021) := (                _sDescription := 'Optimizer',                 _sActiveText := 'Utkoblet',                 _sInactiveText := 'Innkoblet'           );
  A_360_01_SQ5_C411_A1 : FbBinaryInput_Large (2042) := (                _sDescription := 'Luftmengde Sjeld',                 _sActiveText := 'Feil på luftmengde',                 _sInactiveText := 'Ingen feil',                 _udiNotificationClass := 22           );
  A_360_01_SQ5_C411_A2 : FbBinaryInput_Large (2043) := (                _sDescription := 'Kommunikasjonovervåking',                 _sActiveText := 'Kommunikasjonsfeil',                 _sInactiveText := 'Ingen feil',                 _udiNotificationClass := 22           );
  A_360_01_SK5_A421_VOL : FbAnalogInput_Medium (2044) := (                _sDescription := 'Faktisk luftmengde',                 _rCov_Increment := 1,                 _eUnits := WagoTypesBacnet.eBACnetUnits.UNIT_CUBIC_METERS_PER_HOUR           );
  A_360_01_SK5_A421_SP : FbAnalogValue_Medium (2066) := (                _sDescription := 'Settpunkt',                 _rCov_Increment := 1,                 _eUnits := WagoTypesBacnet.eBACnetUnits.UNIT_CUBIC_METERS_PER_HOUR           );
  A_360_01_SK5_A421_VMIN : FbAnalogValue_Medium (2067) := (                _sDescription := 'Minste luftmengde',                 _rCov_Increment := 1,                 _eUnits := WagoTypesBacnet.eBACnetUnits.UNIT_CUBIC_METERS_PER_HOUR           );
  A_360_01_SK5_A421_VMAX : FbAnalogValue_Medium (2068) := (                _sDescription := 'Største luftmengde',                 _rCov_Increment := 1,                 _eUnits := WagoTypesBacnet.eBACnetUnits.UNIT_CUBIC_METERS_PER_HOUR           );
  A_360_01_SK5_A421_FB : FbAnalogInput_Medium (2045) := (                _sDescription := 'Spjeldvinkel',                 _rCov_Increment := 1,                 _eUnits := WagoTypesBacnet.eBACnetUnits.UNIT_PERCENT           );
  A_360_01_SK5_A421_C : FbAnalogOutput_Medium (2022) := (                _sDescription := 'Pådrag',                 _rCov_Increment := 1,                 _eUnits := WagoTypesBacnet.eBACnetUnits.UNIT_PERCENT           );
  A_360_01_SK5_A421_KMD : FbMultiStateValue_Large (2022) := (                _sDescription := 'Manuell overstyring',                 _udiNumberOfStates := 8           );
  A_360_01_SK5_A421_OPT_EKSKL : FbBinaryValue_Medium (2022) := (                _sDescription := 'Optimizer',                 _sActiveText := 'Utkoblet',                 _sInactiveText := 'Innkoblet'           );
  A_360_01_SK5_A421_A1 : FbBinaryInput_Large (2044) := (                _sDescription := 'Luftmengde Sjeld',                 _sActiveText := 'Feil på luftmengde',                 _sInactiveText := 'Ingen feil',                 _udiNotificationClass := 22           );
  A_360_01_SK5_A421_A2 : FbBinaryInput_Large (2045) := (                _sDescription := 'Kommunikasjonovervåking',                 _sActiveText := 'Kommunikasjonsfeil',                 _sInactiveText := 'Ingen feil',                 _udiNotificationClass := 22           );
  A_360_01_SQ5_4AH2_VOL : FbAnalogInput_Medium (2046) := (                _sDescription := 'Faktisk luftmengde',                 _rCov_Increment := 1,                 _eUnits := WagoTypesBacnet.eBACnetUnits.UNIT_CUBIC_METERS_PER_HOUR           );
  A_360_01_SQ5_4AH2_SP : FbAnalogValue_Medium (2069) := (                _sDescription := 'Settpunkt',                 _rCov_Increment := 1,                 _eUnits := WagoTypesBacnet.eBACnetUnits.UNIT_CUBIC_METERS_PER_HOUR           );
  A_360_01_SQ5_4AH2_VMIN : FbAnalogValue_Medium (2070) := (                _sDescription := 'Minste luftmengde',                 _rCov_Increment := 1,                 _eUnits := WagoTypesBacnet.eBACnetUnits.UNIT_CUBIC_METERS_PER_HOUR           );
  A_360_01_SQ5_4AH2_VMAX : FbAnalogValue_Medium (2071) := (                _sDescription := 'Største luftmengde',                 _rCov_Increment := 1,                 _eUnits := WagoTypesBacnet.eBACnetUnits.UNIT_CUBIC_METERS_PER_HOUR           );
  A_360_01_SQ5_4AH2_FB : FbAnalogInput_Medium (2047) := (                _sDescription := 'Spjeldvinkel',                 _rCov_Increment := 1,                 _eUnits := WagoTypesBacnet.eBACnetUnits.UNIT_PERCENT           );
  A_360_01_SQ5_4AH2_C : FbAnalogOutput_Medium (2023) := (                _sDescription := 'Pådrag',                 _rCov_Increment := 1,                 _eUnits := WagoTypesBacnet.eBACnetUnits.UNIT_PERCENT           );
  A_360_01_SQ5_4AH2_KMD : FbMultiStateValue_Large (2023) := (                _sDescription := 'Manuell overstyring',                 _udiNumberOfStates := 8           );
  A_360_01_SQ5_4AH2_OPT_EKSKL : FbBinaryValue_Medium (2023) := (                _sDescription := 'Optimizer',                 _sActiveText := 'Utkoblet',                 _sInactiveText := 'Innkoblet'           );
  A_360_01_SQ5_4AH2_A1 : FbBinaryInput_Large (2046) := (                _sDescription := 'Luftmengde Sjeld',                 _sActiveText := 'Feil på luftmengde',                 _sInactiveText := 'Ingen feil',                 _udiNotificationClass := 22           );
  A_360_01_SQ5_4AH2_A2 : FbBinaryInput_Large (2047) := (                _sDescription := 'Kommunikasjonovervåking',                 _sActiveText := 'Kommunikasjonsfeil',                 _sInactiveText := 'Ingen feil',                 _udiNotificationClass := 22           );
  A_360_01_SK5_A424_VOL : FbAnalogInput_Medium (2048) := (                _sDescription := 'Faktisk luftmengde',                 _rCov_Increment := 1,                 _eUnits := WagoTypesBacnet.eBACnetUnits.UNIT_CUBIC_METERS_PER_HOUR           );
  A_360_01_SK5_A424_SP : FbAnalogValue_Medium (2072) := (                _sDescription := 'Settpunkt',                 _rCov_Increment := 1,                 _eUnits := WagoTypesBacnet.eBACnetUnits.UNIT_CUBIC_METERS_PER_HOUR           );
  A_360_01_SK5_A424_VMIN : FbAnalogValue_Medium (2073) := (                _sDescription := 'Minste luftmengde',                 _rCov_Increment := 1,                 _eUnits := WagoTypesBacnet.eBACnetUnits.UNIT_CUBIC_METERS_PER_HOUR           );
  A_360_01_SK5_A424_VMAX : FbAnalogValue_Medium (2074) := (                _sDescription := 'Største luftmengde',                 _rCov_Increment := 1,                 _eUnits := WagoTypesBacnet.eBACnetUnits.UNIT_CUBIC_METERS_PER_HOUR           );
  A_360_01_SK5_A424_FB : FbAnalogInput_Medium (2049) := (                _sDescription := 'Spjeldvinkel',                 _rCov_Increment := 1,                 _eUnits := WagoTypesBacnet.eBACnetUnits.UNIT_PERCENT           );
  A_360_01_SK5_A424_C : FbAnalogOutput_Medium (2024) := (                _sDescription := 'Pådrag',                 _rCov_Increment := 1,                 _eUnits := WagoTypesBacnet.eBACnetUnits.UNIT_PERCENT           );
  A_360_01_SK5_A424_KMD : FbMultiStateValue_Large (2024) := (                _sDescription := 'Manuell overstyring',                 _udiNumberOfStates := 8           );
  A_360_01_SK5_A424_OPT_EKSKL : FbBinaryValue_Medium (2024) := (                _sDescription := 'Optimizer',                 _sActiveText := 'Utkoblet',                 _sInactiveText := 'Innkoblet'           );
  A_360_01_SK5_A424_A1 : FbBinaryInput_Large (2048) := (                _sDescription := 'Luftmengde Sjeld',                 _sActiveText := 'Feil på luftmengde',                 _sInactiveText := 'Ingen feil',                 _udiNotificationClass := 22           );
  A_360_01_SK5_A424_A2 : FbBinaryInput_Large (2049) := (                _sDescription := 'Kommunikasjonovervåking',                 _sActiveText := 'Kommunikasjonsfeil',                 _sInactiveText := 'Ingen feil',                 _udiNotificationClass := 22           );
  A_360_01_SQ4_4AH3_VOL : FbAnalogInput_Medium (2050) := (                _sDescription := 'Faktisk luftmengde',                 _rCov_Increment := 1,                 _eUnits := WagoTypesBacnet.eBACnetUnits.UNIT_CUBIC_METERS_PER_HOUR           );
  A_360_01_SQ4_4AH3_SP : FbAnalogValue_Medium (2075) := (                _sDescription := 'Settpunkt',                 _rCov_Increment := 1,                 _eUnits := WagoTypesBacnet.eBACnetUnits.UNIT_CUBIC_METERS_PER_HOUR           );
  A_360_01_SQ4_4AH3_VMIN : FbAnalogValue_Medium (2076) := (                _sDescription := 'Minste luftmengde',                 _rCov_Increment := 1,                 _eUnits := WagoTypesBacnet.eBACnetUnits.UNIT_CUBIC_METERS_PER_HOUR           );
  A_360_01_SQ4_4AH3_VMAX : FbAnalogValue_Medium (2077) := (                _sDescription := 'Største luftmengde',                 _rCov_Increment := 1,                 _eUnits := WagoTypesBacnet.eBACnetUnits.UNIT_CUBIC_METERS_PER_HOUR           );
  A_360_01_SQ4_4AH3_FB : FbAnalogInput_Medium (2051) := (                _sDescription := 'Spjeldvinkel',                 _rCov_Increment := 1,                 _eUnits := WagoTypesBacnet.eBACnetUnits.UNIT_PERCENT           );
  A_360_01_SQ4_4AH3_C : FbAnalogOutput_Medium (2025) := (                _sDescription := 'Pådrag',                 _rCov_Increment := 1,                 _eUnits := WagoTypesBacnet.eBACnetUnits.UNIT_PERCENT           );
  A_360_01_SQ4_4AH3_KMD : FbMultiStateValue_Large (2025) := (                _sDescription := 'Manuell overstyring',                 _udiNumberOfStates := 8           );
  A_360_01_SQ4_4AH3_OPT_EKSKL : FbBinaryValue_Medium (2025) := (                _sDescription := 'Optimizer',                 _sActiveText := 'Utkoblet',                 _sInactiveText := 'Innkoblet'           );
  A_360_01_SQ4_4AH3_A1 : FbBinaryInput_Large (2050) := (                _sDescription := 'Luftmengde Sjeld',                 _sActiveText := 'Feil på luftmengde',                 _sInactiveText := 'Ingen feil',                 _udiNotificationClass := 22           );
  A_360_01_SQ4_4AH3_A2 : FbBinaryInput_Large (2051) := (                _sDescription := 'Kommunikasjonovervåking',                 _sActiveText := 'Kommunikasjonsfeil',                 _sInactiveText := 'Ingen feil',                 _udiNotificationClass := 22           );
  A_360_01_SQ4_4AH4_VOL : FbAnalogInput_Medium (2052) := (                _sDescription := 'Faktisk luftmengde',                 _rCov_Increment := 1,                 _eUnits := WagoTypesBacnet.eBACnetUnits.UNIT_CUBIC_METERS_PER_HOUR           );
  A_360_01_SQ4_4AH4_SP : FbAnalogValue_Medium (2078) := (                _sDescription := 'Settpunkt',                 _rCov_Increment := 1,                 _eUnits := WagoTypesBacnet.eBACnetUnits.UNIT_CUBIC_METERS_PER_HOUR           );
  A_360_01_SQ4_4AH4_VMIN : FbAnalogValue_Medium (2079) := (                _sDescription := 'Minste luftmengde',                 _rCov_Increment := 1,                 _eUnits := WagoTypesBacnet.eBACnetUnits.UNIT_CUBIC_METERS_PER_HOUR           );
  A_360_01_SQ4_4AH4_VMAX : FbAnalogValue_Medium (2080) := (                _sDescription := 'Største luftmengde',                 _rCov_Increment := 1,                 _eUnits := WagoTypesBacnet.eBACnetUnits.UNIT_CUBIC_METERS_PER_HOUR           );
  A_360_01_SQ4_4AH4_FB : FbAnalogInput_Medium (2053) := (                _sDescription := 'Spjeldvinkel',                 _rCov_Increment := 1,                 _eUnits := WagoTypesBacnet.eBACnetUnits.UNIT_PERCENT           );
  A_360_01_SQ4_4AH4_C : FbAnalogOutput_Medium (2026) := (                _sDescription := 'Pådrag',                 _rCov_Increment := 1,                 _eUnits := WagoTypesBacnet.eBACnetUnits.UNIT_PERCENT           );
  A_360_01_SQ4_4AH4_KMD : FbMultiStateValue_Large (2026) := (                _sDescription := 'Manuell overstyring',                 _udiNumberOfStates := 8           );
  A_360_01_SQ4_4AH4_OPT_EKSKL : FbBinaryValue_Medium (2026) := (                _sDescription := 'Optimizer',                 _sActiveText := 'Utkoblet',                 _sInactiveText := 'Innkoblet'           );
  A_360_01_SQ4_4AH4_A1 : FbBinaryInput_Large (2052) := (                _sDescription := 'Luftmengde Sjeld',                 _sActiveText := 'Feil på luftmengde',                 _sInactiveText := 'Ingen feil',                 _udiNotificationClass := 22           );
  A_360_01_SQ4_4AH4_A2 : FbBinaryInput_Large (2053) := (                _sDescription := 'Kommunikasjonovervåking',                 _sActiveText := 'Kommunikasjonsfeil',                 _sInactiveText := 'Ingen feil',                 _udiNotificationClass := 22           );
  A_360_01_SQ4_4AH5_VOL : FbAnalogInput_Medium (2054) := (                _sDescription := 'Faktisk luftmengde',                 _rCov_Increment := 1,                 _eUnits := WagoTypesBacnet.eBACnetUnits.UNIT_CUBIC_METERS_PER_HOUR           );
  A_360_01_SQ4_4AH5_SP : FbAnalogValue_Medium (2081) := (                _sDescription := 'Settpunkt',                 _rCov_Increment := 1,                 _eUnits := WagoTypesBacnet.eBACnetUnits.UNIT_CUBIC_METERS_PER_HOUR           );
  A_360_01_SQ4_4AH5_VMIN : FbAnalogValue_Medium (2082) := (                _sDescription := 'Minste luftmengde',                 _rCov_Increment := 1,                 _eUnits := WagoTypesBacnet.eBACnetUnits.UNIT_CUBIC_METERS_PER_HOUR           );
  A_360_01_SQ4_4AH5_VMAX : FbAnalogValue_Medium (2083) := (                _sDescription := 'Største luftmengde',                 _rCov_Increment := 1,                 _eUnits := WagoTypesBacnet.eBACnetUnits.UNIT_CUBIC_METERS_PER_HOUR           );
  A_360_01_SQ4_4AH5_FB : FbAnalogInput_Medium (2055) := (                _sDescription := 'Spjeldvinkel',                 _rCov_Increment := 1,                 _eUnits := WagoTypesBacnet.eBACnetUnits.UNIT_PERCENT           );
  A_360_01_SQ4_4AH5_C : FbAnalogOutput_Medium (2027) := (                _sDescription := 'Pådrag',                 _rCov_Increment := 1,                 _eUnits := WagoTypesBacnet.eBACnetUnits.UNIT_PERCENT           );
  A_360_01_SQ4_4AH5_KMD : FbMultiStateValue_Large (2027) := (                _sDescription := 'Manuell overstyring',                 _udiNumberOfStates := 8           );
  A_360_01_SQ4_4AH5_OPT_EKSKL : FbBinaryValue_Medium (2027) := (                _sDescription := 'Optimizer',                 _sActiveText := 'Utkoblet',                 _sInactiveText := 'Innkoblet'           );
  A_360_01_SQ4_4AH5_A1 : FbBinaryInput_Large (2054) := (                _sDescription := 'Luftmengde Sjeld',                 _sActiveText := 'Feil på luftmengde',                 _sInactiveText := 'Ingen feil',                 _udiNotificationClass := 22           );
  A_360_01_SQ4_4AH5_A2 : FbBinaryInput_Large (2055) := (                _sDescription := 'Kommunikasjonovervåking',                 _sActiveText := 'Kommunikasjonsfeil',                 _sInactiveText := 'Ingen feil',                 _udiNotificationClass := 22           );
  A_360_01_SQ5_4AH3_VOL : FbAnalogInput_Medium (2056) := (                _sDescription := 'Faktisk luftmengde',                 _rCov_Increment := 1,                 _eUnits := WagoTypesBacnet.eBACnetUnits.UNIT_CUBIC_METERS_PER_HOUR           );
  A_360_01_SQ5_4AH3_SP : FbAnalogValue_Medium (2084) := (                _sDescription := 'Settpunkt',                 _rCov_Increment := 1,                 _eUnits := WagoTypesBacnet.eBACnetUnits.UNIT_CUBIC_METERS_PER_HOUR           );
  A_360_01_SQ5_4AH3_VMIN : FbAnalogValue_Medium (2085) := (                _sDescription := 'Minste luftmengde',                 _rCov_Increment := 1,                 _eUnits := WagoTypesBacnet.eBACnetUnits.UNIT_CUBIC_METERS_PER_HOUR           );
  A_360_01_SQ5_4AH3_VMAX : FbAnalogValue_Medium (2086) := (                _sDescription := 'Største luftmengde',                 _rCov_Increment := 1,                 _eUnits := WagoTypesBacnet.eBACnetUnits.UNIT_CUBIC_METERS_PER_HOUR           );
  A_360_01_SQ5_4AH3_FB : FbAnalogInput_Medium (2057) := (                _sDescription := 'Spjeldvinkel',                 _rCov_Increment := 1,                 _eUnits := WagoTypesBacnet.eBACnetUnits.UNIT_PERCENT           );
  A_360_01_SQ5_4AH3_C : FbAnalogOutput_Medium (2028) := (                _sDescription := 'Pådrag',                 _rCov_Increment := 1,                 _eUnits := WagoTypesBacnet.eBACnetUnits.UNIT_PERCENT           );
  A_360_01_SQ5_4AH3_KMD : FbMultiStateValue_Large (2028) := (                _sDescription := 'Manuell overstyring',                 _udiNumberOfStates := 8           );
  A_360_01_SQ5_4AH3_OPT_EKSKL : FbBinaryValue_Medium (2028) := (                _sDescription := 'Optimizer',                 _sActiveText := 'Utkoblet',                 _sInactiveText := 'Innkoblet'           );
  A_360_01_SQ5_4AH3_A1 : FbBinaryInput_Large (2056) := (                _sDescription := 'Luftmengde Sjeld',                 _sActiveText := 'Feil på luftmengde',                 _sInactiveText := 'Ingen feil',                 _udiNotificationClass := 22           );
  A_360_01_SQ5_4AH3_A2 : FbBinaryInput_Large (2057) := (                _sDescription := 'Kommunikasjonovervåking',                 _sActiveText := 'Kommunikasjonsfeil',                 _sInactiveText := 'Ingen feil',                 _udiNotificationClass := 22           );
  A_360_01_SQ5_A401_VOL : FbAnalogInput_Medium (2058) := (                _sDescription := 'Faktisk luftmengde',                 _rCov_Increment := 1,                 _eUnits := WagoTypesBacnet.eBACnetUnits.UNIT_CUBIC_METERS_PER_HOUR           );
  A_360_01_SQ5_A401_SP : FbAnalogValue_Medium (2087) := (                _sDescription := 'Settpunkt',                 _rCov_Increment := 1,                 _eUnits := WagoTypesBacnet.eBACnetUnits.UNIT_CUBIC_METERS_PER_HOUR           );
  A_360_01_SQ5_A401_VMIN : FbAnalogValue_Medium (2088) := (                _sDescription := 'Minste luftmengde',                 _rCov_Increment := 1,                 _eUnits := WagoTypesBacnet.eBACnetUnits.UNIT_CUBIC_METERS_PER_HOUR           );
  A_360_01_SQ5_A401_VMAX : FbAnalogValue_Medium (2089) := (                _sDescription := 'Største luftmengde',                 _rCov_Increment := 1,                 _eUnits := WagoTypesBacnet.eBACnetUnits.UNIT_CUBIC_METERS_PER_HOUR           );
  A_360_01_SQ5_A401_FB : FbAnalogInput_Medium (2059) := (                _sDescription := 'Spjeldvinkel',                 _rCov_Increment := 1,                 _eUnits := WagoTypesBacnet.eBACnetUnits.UNIT_PERCENT           );
  A_360_01_SQ5_A401_C : FbAnalogOutput_Medium (2029) := (                _sDescription := 'Pådrag',                 _rCov_Increment := 1,                 _eUnits := WagoTypesBacnet.eBACnetUnits.UNIT_PERCENT           );
  A_360_01_SQ5_A401_KMD : FbMultiStateValue_Large (2029) := (                _sDescription := 'Manuell overstyring',                 _udiNumberOfStates := 8           );
  A_360_01_SQ5_A401_OPT_EKSKL : FbBinaryValue_Medium (2029) := (                _sDescription := 'Optimizer',                 _sActiveText := 'Utkoblet',                 _sInactiveText := 'Innkoblet'           );
  A_360_01_SQ5_A401_A1 : FbBinaryInput_Large (2058) := (                _sDescription := 'Luftmengde Sjeld',                 _sActiveText := 'Feil på luftmengde',                 _sInactiveText := 'Ingen feil',                 _udiNotificationClass := 22           );
  A_360_01_SQ5_A401_A2 : FbBinaryInput_Large (2059) := (                _sDescription := 'Kommunikasjonovervåking',                 _sActiveText := 'Kommunikasjonsfeil',                 _sInactiveText := 'Ingen feil',                 _udiNotificationClass := 22           );
  A_360_01_SQ4_A403_VOL : FbAnalogInput_Medium (2060) := (                _sDescription := 'Faktisk luftmengde',                 _rCov_Increment := 1,                 _eUnits := WagoTypesBacnet.eBACnetUnits.UNIT_CUBIC_METERS_PER_HOUR           );
  A_360_01_SQ4_A403_SP : FbAnalogValue_Medium (2090) := (                _sDescription := 'Settpunkt',                 _rCov_Increment := 1,                 _eUnits := WagoTypesBacnet.eBACnetUnits.UNIT_CUBIC_METERS_PER_HOUR           );
  A_360_01_SQ4_A403_VMIN : FbAnalogValue_Medium (2091) := (                _sDescription := 'Minste luftmengde',                 _rCov_Increment := 1,                 _eUnits := WagoTypesBacnet.eBACnetUnits.UNIT_CUBIC_METERS_PER_HOUR           );
  A_360_01_SQ4_A403_VMAX : FbAnalogValue_Medium (2092) := (                _sDescription := 'Største luftmengde',                 _rCov_Increment := 1,                 _eUnits := WagoTypesBacnet.eBACnetUnits.UNIT_CUBIC_METERS_PER_HOUR           );
  A_360_01_SQ4_A403_FB : FbAnalogInput_Medium (2061) := (                _sDescription := 'Spjeldvinkel',                 _rCov_Increment := 1,                 _eUnits := WagoTypesBacnet.eBACnetUnits.UNIT_PERCENT           );
  A_360_01_SQ4_A403_C : FbAnalogOutput_Medium (2030) := (                _sDescription := 'Pådrag',                 _rCov_Increment := 1,                 _eUnits := WagoTypesBacnet.eBACnetUnits.UNIT_PERCENT           );
  A_360_01_SQ4_A403_KMD : FbMultiStateValue_Large (2030) := (                _sDescription := 'Manuell overstyring',                 _udiNumberOfStates := 8           );
  A_360_01_SQ4_A403_OPT_EKSKL : FbBinaryValue_Medium (2030) := (                _sDescription := 'Optimizer',                 _sActiveText := 'Utkoblet',                 _sInactiveText := 'Innkoblet'           );
  A_360_01_SQ4_A403_A1 : FbBinaryInput_Large (2060) := (                _sDescription := 'Luftmengde Sjeld',                 _sActiveText := 'Feil på luftmengde',                 _sInactiveText := 'Ingen feil',                 _udiNotificationClass := 22           );
  A_360_01_SQ4_A403_A2 : FbBinaryInput_Large (2061) := (                _sDescription := 'Kommunikasjonovervåking',                 _sActiveText := 'Kommunikasjonsfeil',                 _sInactiveText := 'Ingen feil',                 _udiNotificationClass := 22           );
  A_360_01_SQ4_A401_3_VOL : FbAnalogInput_Medium (2062) := (                _sDescription := 'Faktisk luftmengde',                 _rCov_Increment := 1,                 _eUnits := WagoTypesBacnet.eBACnetUnits.UNIT_CUBIC_METERS_PER_HOUR           );
  A_360_01_SQ4_A401_3_SP : FbAnalogValue_Medium (2093) := (                _sDescription := 'Settpunkt',                 _rCov_Increment := 1,                 _eUnits := WagoTypesBacnet.eBACnetUnits.UNIT_CUBIC_METERS_PER_HOUR           );
  A_360_01_SQ4_A401_3_VMIN : FbAnalogValue_Medium (2094) := (                _sDescription := 'Minste luftmengde',                 _rCov_Increment := 1,                 _eUnits := WagoTypesBacnet.eBACnetUnits.UNIT_CUBIC_METERS_PER_HOUR           );
  A_360_01_SQ4_A401_3_VMAX : FbAnalogValue_Medium (2095) := (                _sDescription := 'Største luftmengde',                 _rCov_Increment := 1,                 _eUnits := WagoTypesBacnet.eBACnetUnits.UNIT_CUBIC_METERS_PER_HOUR           );
  A_360_01_SQ4_A401_3_FB : FbAnalogInput_Medium (2063) := (                _sDescription := 'Spjeldvinkel',                 _rCov_Increment := 1,                 _eUnits := WagoTypesBacnet.eBACnetUnits.UNIT_PERCENT           );
  A_360_01_SQ4_A401_3_C : FbAnalogOutput_Medium (2031) := (                _sDescription := 'Pådrag',                 _rCov_Increment := 1,                 _eUnits := WagoTypesBacnet.eBACnetUnits.UNIT_PERCENT           );
  A_360_01_SQ4_A401_3_KMD : FbMultiStateValue_Large (2031) := (                _sDescription := 'Manuell overstyring',                 _udiNumberOfStates := 8           );
  A_360_01_SQ4_A401_3_OPT_EKSKL : FbBinaryValue_Medium (2031) := (                _sDescription := 'Optimizer',                 _sActiveText := 'Utkoblet',                 _sInactiveText := 'Innkoblet'           );
  A_360_01_SQ4_A401_3_A1 : FbBinaryInput_Large (2062) := (                _sDescription := 'Luftmengde Sjeld',                 _sActiveText := 'Feil på luftmengde',                 _sInactiveText := 'Ingen feil',                 _udiNotificationClass := 22           );
  A_360_01_SQ4_A401_3_A2 : FbBinaryInput_Large (2063) := (                _sDescription := 'Kommunikasjonovervåking',                 _sActiveText := 'Kommunikasjonsfeil',                 _sInactiveText := 'Ingen feil',                 _udiNotificationClass := 22           );
  A_360_01_SQ4_A401_4_VOL : FbAnalogInput_Medium (2064) := (                _sDescription := 'Faktisk luftmengde',                 _rCov_Increment := 1,                 _eUnits := WagoTypesBacnet.eBACnetUnits.UNIT_CUBIC_METERS_PER_HOUR           );
  A_360_01_SQ4_A401_4_SP : FbAnalogValue_Medium (2096) := (                _sDescription := 'Settpunkt',                 _rCov_Increment := 1,                 _eUnits := WagoTypesBacnet.eBACnetUnits.UNIT_CUBIC_METERS_PER_HOUR           );
  A_360_01_SQ4_A401_4_VMIN : FbAnalogValue_Medium (2097) := (                _sDescription := 'Minste luftmengde',                 _rCov_Increment := 1,                 _eUnits := WagoTypesBacnet.eBACnetUnits.UNIT_CUBIC_METERS_PER_HOUR           );
  A_360_01_SQ4_A401_4_VMAX : FbAnalogValue_Medium (2098) := (                _sDescription := 'Største luftmengde',                 _rCov_Increment := 1,                 _eUnits := WagoTypesBacnet.eBACnetUnits.UNIT_CUBIC_METERS_PER_HOUR           );
  A_360_01_SQ4_A401_4_FB : FbAnalogInput_Medium (2065) := (                _sDescription := 'Spjeldvinkel',                 _rCov_Increment := 1,                 _eUnits := WagoTypesBacnet.eBACnetUnits.UNIT_PERCENT           );
  A_360_01_SQ4_A401_4_C : FbAnalogOutput_Medium (2032) := (                _sDescription := 'Pådrag',                 _rCov_Increment := 1,                 _eUnits := WagoTypesBacnet.eBACnetUnits.UNIT_PERCENT           );
  A_360_01_SQ4_A401_4_KMD : FbMultiStateValue_Large (2032) := (                _sDescription := 'Manuell overstyring',                 _udiNumberOfStates := 8           );
  A_360_01_SQ4_A401_4_OPT_EKSKL : FbBinaryValue_Medium (2032) := (                _sDescription := 'Optimizer',                 _sActiveText := 'Utkoblet',                 _sInactiveText := 'Innkoblet'           );
  A_360_01_SQ4_A401_4_A1 : FbBinaryInput_Large (2064) := (                _sDescription := 'Luftmengde Sjeld',                 _sActiveText := 'Feil på luftmengde',                 _sInactiveText := 'Ingen feil',                 _udiNotificationClass := 22           );
  A_360_01_SQ4_A401_4_A2 : FbBinaryInput_Large (2065) := (                _sDescription := 'Kommunikasjonovervåking',                 _sActiveText := 'Kommunikasjonsfeil',                 _sInactiveText := 'Ingen feil',                 _udiNotificationClass := 22           );
  A_360_01_SQ4_A401_5_VOL : FbAnalogInput_Medium (2066) := (                _sDescription := 'Faktisk luftmengde',                 _rCov_Increment := 1,                 _eUnits := WagoTypesBacnet.eBACnetUnits.UNIT_CUBIC_METERS_PER_HOUR           );
  A_360_01_SQ4_A401_5_SP : FbAnalogValue_Medium (2099) := (                _sDescription := 'Settpunkt',                 _rCov_Increment := 1,                 _eUnits := WagoTypesBacnet.eBACnetUnits.UNIT_CUBIC_METERS_PER_HOUR           );
  A_360_01_SQ4_A401_5_VMIN : FbAnalogValue_Medium (2100) := (                _sDescription := 'Minste luftmengde',                 _rCov_Increment := 1,                 _eUnits := WagoTypesBacnet.eBACnetUnits.UNIT_CUBIC_METERS_PER_HOUR           );
  A_360_01_SQ4_A401_5_VMAX : FbAnalogValue_Medium (2101) := (                _sDescription := 'Største luftmengde',                 _rCov_Increment := 1,                 _eUnits := WagoTypesBacnet.eBACnetUnits.UNIT_CUBIC_METERS_PER_HOUR           );
  A_360_01_SQ4_A401_5_FB : FbAnalogInput_Medium (2067) := (                _sDescription := 'Spjeldvinkel',                 _rCov_Increment := 1,                 _eUnits := WagoTypesBacnet.eBACnetUnits.UNIT_PERCENT           );
  A_360_01_SQ4_A401_5_C : FbAnalogOutput_Medium (2033) := (                _sDescription := 'Pådrag',                 _rCov_Increment := 1,                 _eUnits := WagoTypesBacnet.eBACnetUnits.UNIT_PERCENT           );
  A_360_01_SQ4_A401_5_KMD : FbMultiStateValue_Large (2033) := (                _sDescription := 'Manuell overstyring',                 _udiNumberOfStates := 8           );
  A_360_01_SQ4_A401_5_OPT_EKSKL : FbBinaryValue_Medium (2033) := (                _sDescription := 'Optimizer',                 _sActiveText := 'Utkoblet',                 _sInactiveText := 'Innkoblet'           );
  A_360_01_SQ4_A401_5_A1 : FbBinaryInput_Large (2066) := (                _sDescription := 'Luftmengde Sjeld',                 _sActiveText := 'Feil på luftmengde',                 _sInactiveText := 'Ingen feil',                 _udiNotificationClass := 22           );
  A_360_01_SQ4_A401_5_A2 : FbBinaryInput_Large (2067) := (                _sDescription := 'Kommunikasjonovervåking',                 _sActiveText := 'Kommunikasjonsfeil',                 _sInactiveText := 'Ingen feil',                 _udiNotificationClass := 22           );
  A_360_01_SQ4_A401_6_VOL : FbAnalogInput_Medium (2068) := (                _sDescription := 'Faktisk luftmengde',                 _rCov_Increment := 1,                 _eUnits := WagoTypesBacnet.eBACnetUnits.UNIT_CUBIC_METERS_PER_HOUR           );
  A_360_01_SQ4_A401_6_SP : FbAnalogValue_Medium (2102) := (                _sDescription := 'Settpunkt',                 _rCov_Increment := 1,                 _eUnits := WagoTypesBacnet.eBACnetUnits.UNIT_CUBIC_METERS_PER_HOUR           );
  A_360_01_SQ4_A401_6_VMIN : FbAnalogValue_Medium (2103) := (                _sDescription := 'Minste luftmengde',                 _rCov_Increment := 1,                 _eUnits := WagoTypesBacnet.eBACnetUnits.UNIT_CUBIC_METERS_PER_HOUR           );
  A_360_01_SQ4_A401_6_VMAX : FbAnalogValue_Medium (2104) := (                _sDescription := 'Største luftmengde',                 _rCov_Increment := 1,                 _eUnits := WagoTypesBacnet.eBACnetUnits.UNIT_CUBIC_METERS_PER_HOUR           );
  A_360_01_SQ4_A401_6_FB : FbAnalogInput_Medium (2069) := (                _sDescription := 'Spjeldvinkel',                 _rCov_Increment := 1,                 _eUnits := WagoTypesBacnet.eBACnetUnits.UNIT_PERCENT           );
  A_360_01_SQ4_A401_6_C : FbAnalogOutput_Medium (2034) := (                _sDescription := 'Pådrag',                 _rCov_Increment := 1,                 _eUnits := WagoTypesBacnet.eBACnetUnits.UNIT_PERCENT           );
  A_360_01_SQ4_A401_6_KMD : FbMultiStateValue_Large (2034) := (                _sDescription := 'Manuell overstyring',                 _udiNumberOfStates := 8           );
  A_360_01_SQ4_A401_6_OPT_EKSKL : FbBinaryValue_Medium (2034) := (                _sDescription := 'Optimizer',                 _sActiveText := 'Utkoblet',                 _sInactiveText := 'Innkoblet'           );
  A_360_01_SQ4_A401_6_A1 : FbBinaryInput_Large (2068) := (                _sDescription := 'Luftmengde Sjeld',                 _sActiveText := 'Feil på luftmengde',                 _sInactiveText := 'Ingen feil',                 _udiNotificationClass := 22           );
  A_360_01_SQ4_A401_6_A2 : FbBinaryInput_Large (2069) := (                _sDescription := 'Kommunikasjonovervåking',                 _sActiveText := 'Kommunikasjonsfeil',                 _sInactiveText := 'Ingen feil',                 _udiNotificationClass := 22           );
  A_360_01_SQ4_A401_7_VOL : FbAnalogInput_Medium (2070) := (                _sDescription := 'Faktisk luftmengde',                 _rCov_Increment := 1,                 _eUnits := WagoTypesBacnet.eBACnetUnits.UNIT_CUBIC_METERS_PER_HOUR           );
  A_360_01_SQ4_A401_7_SP : FbAnalogValue_Medium (2105) := (                _sDescription := 'Settpunkt',                 _rCov_Increment := 1,                 _eUnits := WagoTypesBacnet.eBACnetUnits.UNIT_CUBIC_METERS_PER_HOUR           );
  A_360_01_SQ4_A401_7_VMIN : FbAnalogValue_Medium (2106) := (                _sDescription := 'Minste luftmengde',                 _rCov_Increment := 1,                 _eUnits := WagoTypesBacnet.eBACnetUnits.UNIT_CUBIC_METERS_PER_HOUR           );
  A_360_01_SQ4_A401_7_VMAX : FbAnalogValue_Medium (2107) := (                _sDescription := 'Største luftmengde',                 _rCov_Increment := 1,                 _eUnits := WagoTypesBacnet.eBACnetUnits.UNIT_CUBIC_METERS_PER_HOUR           );
  A_360_01_SQ4_A401_7_FB : FbAnalogInput_Medium (2071) := (                _sDescription := 'Spjeldvinkel',                 _rCov_Increment := 1,                 _eUnits := WagoTypesBacnet.eBACnetUnits.UNIT_PERCENT           );
  A_360_01_SQ4_A401_7_C : FbAnalogOutput_Medium (2035) := (                _sDescription := 'Pådrag',                 _rCov_Increment := 1,                 _eUnits := WagoTypesBacnet.eBACnetUnits.UNIT_PERCENT           );
  A_360_01_SQ4_A401_7_KMD : FbMultiStateValue_Large (2035) := (                _sDescription := 'Manuell overstyring',                 _udiNumberOfStates := 8           );
  A_360_01_SQ4_A401_7_OPT_EKSKL : FbBinaryValue_Medium (2035) := (                _sDescription := 'Optimizer',                 _sActiveText := 'Utkoblet',                 _sInactiveText := 'Innkoblet'           );
  A_360_01_SQ4_A401_7_A1 : FbBinaryInput_Large (2070) := (                _sDescription := 'Luftmengde Sjeld',                 _sActiveText := 'Feil på luftmengde',                 _sInactiveText := 'Ingen feil',                 _udiNotificationClass := 22           );
  A_360_01_SQ4_A401_7_A2 : FbBinaryInput_Large (2071) := (                _sDescription := 'Kommunikasjonovervåking',                 _sActiveText := 'Kommunikasjonsfeil',                 _sInactiveText := 'Ingen feil',                 _udiNotificationClass := 22           );
  A_360_01_SQ4_A401_8_VOL : FbAnalogInput_Medium (2072) := (                _sDescription := 'Faktisk luftmengde',                 _rCov_Increment := 1,                 _eUnits := WagoTypesBacnet.eBACnetUnits.UNIT_CUBIC_METERS_PER_HOUR           );
  A_360_01_SQ4_A401_8_SP : FbAnalogValue_Medium (2108) := (                _sDescription := 'Settpunkt',                 _rCov_Increment := 1,                 _eUnits := WagoTypesBacnet.eBACnetUnits.UNIT_CUBIC_METERS_PER_HOUR           );
  A_360_01_SQ4_A401_8_VMIN : FbAnalogValue_Medium (2109) := (                _sDescription := 'Minste luftmengde',                 _rCov_Increment := 1,                 _eUnits := WagoTypesBacnet.eBACnetUnits.UNIT_CUBIC_METERS_PER_HOUR           );
  A_360_01_SQ4_A401_8_VMAX : FbAnalogValue_Medium (2110) := (                _sDescription := 'Største luftmengde',                 _rCov_Increment := 1,                 _eUnits := WagoTypesBacnet.eBACnetUnits.UNIT_CUBIC_METERS_PER_HOUR           );
  A_360_01_SQ4_A401_8_FB : FbAnalogInput_Medium (2073) := (                _sDescription := 'Spjeldvinkel',                 _rCov_Increment := 1,                 _eUnits := WagoTypesBacnet.eBACnetUnits.UNIT_PERCENT           );
  A_360_01_SQ4_A401_8_C : FbAnalogOutput_Medium (2036) := (                _sDescription := 'Pådrag',                 _rCov_Increment := 1,                 _eUnits := WagoTypesBacnet.eBACnetUnits.UNIT_PERCENT           );
  A_360_01_SQ4_A401_8_KMD : FbMultiStateValue_Large (2036) := (                _sDescription := 'Manuell overstyring',                 _udiNumberOfStates := 8           );
  A_360_01_SQ4_A401_8_OPT_EKSKL : FbBinaryValue_Medium (2036) := (                _sDescription := 'Optimizer',                 _sActiveText := 'Utkoblet',                 _sInactiveText := 'Innkoblet'           );
  A_360_01_SQ4_A401_8_A1 : FbBinaryInput_Large (2072) := (                _sDescription := 'Luftmengde Sjeld',                 _sActiveText := 'Feil på luftmengde',                 _sInactiveText := 'Ingen feil',                 _udiNotificationClass := 22           );
  A_360_01_SQ4_A401_8_A2 : FbBinaryInput_Large (2073) := (                _sDescription := 'Kommunikasjonovervåking',                 _sActiveText := 'Kommunikasjonsfeil',                 _sInactiveText := 'Ingen feil',                 _udiNotificationClass := 22           );
  A_360_01_SQ4_A401_9_VOL : FbAnalogInput_Medium (2074) := (                _sDescription := 'Faktisk luftmengde',                 _rCov_Increment := 1,                 _eUnits := WagoTypesBacnet.eBACnetUnits.UNIT_CUBIC_METERS_PER_HOUR           );
  A_360_01_SQ4_A401_9_SP : FbAnalogValue_Medium (2111) := (                _sDescription := 'Settpunkt',                 _rCov_Increment := 1,                 _eUnits := WagoTypesBacnet.eBACnetUnits.UNIT_CUBIC_METERS_PER_HOUR           );
  A_360_01_SQ4_A401_9_VMIN : FbAnalogValue_Medium (2112) := (                _sDescription := 'Minste luftmengde',                 _rCov_Increment := 1,                 _eUnits := WagoTypesBacnet.eBACnetUnits.UNIT_CUBIC_METERS_PER_HOUR           );
  A_360_01_SQ4_A401_9_VMAX : FbAnalogValue_Medium (2113) := (                _sDescription := 'Største luftmengde',                 _rCov_Increment := 1,                 _eUnits := WagoTypesBacnet.eBACnetUnits.UNIT_CUBIC_METERS_PER_HOUR           );
  A_360_01_SQ4_A401_9_FB : FbAnalogInput_Medium (2075) := (                _sDescription := 'Spjeldvinkel',                 _rCov_Increment := 1,                 _eUnits := WagoTypesBacnet.eBACnetUnits.UNIT_PERCENT           );
  A_360_01_SQ4_A401_9_C : FbAnalogOutput_Medium (2037) := (                _sDescription := 'Pådrag',                 _rCov_Increment := 1,                 _eUnits := WagoTypesBacnet.eBACnetUnits.UNIT_PERCENT           );
  A_360_01_SQ4_A401_9_KMD : FbMultiStateValue_Large (2037) := (                _sDescription := 'Manuell overstyring',                 _udiNumberOfStates := 8           );
  A_360_01_SQ4_A401_9_OPT_EKSKL : FbBinaryValue_Medium (2037) := (                _sDescription := 'Optimizer',                 _sActiveText := 'Utkoblet',                 _sInactiveText := 'Innkoblet'           );
  A_360_01_SQ4_A401_9_A1 : FbBinaryInput_Large (2074) := (                _sDescription := 'Luftmengde Sjeld',                 _sActiveText := 'Feil på luftmengde',                 _sInactiveText := 'Ingen feil',                 _udiNotificationClass := 22           );
  A_360_01_SQ4_A401_9_A2 : FbBinaryInput_Large (2075) := (                _sDescription := 'Kommunikasjonovervåking',                 _sActiveText := 'Kommunikasjonsfeil',                 _sInactiveText := 'Ingen feil',                 _udiNotificationClass := 22           );
  A_360_01_SQ4_A401_0_VOL : FbAnalogInput_Medium (2076) := (                _sDescription := 'Faktisk luftmengde',                 _rCov_Increment := 1,                 _eUnits := WagoTypesBacnet.eBACnetUnits.UNIT_CUBIC_METERS_PER_HOUR           );
  A_360_01_SQ4_A401_0_SP : FbAnalogValue_Medium (2114) := (                _sDescription := 'Settpunkt',                 _rCov_Increment := 1,                 _eUnits := WagoTypesBacnet.eBACnetUnits.UNIT_CUBIC_METERS_PER_HOUR           );
  A_360_01_SQ4_A401_0_VMIN : FbAnalogValue_Medium (2115) := (                _sDescription := 'Minste luftmengde',                 _rCov_Increment := 1,                 _eUnits := WagoTypesBacnet.eBACnetUnits.UNIT_CUBIC_METERS_PER_HOUR           );
  A_360_01_SQ4_A401_0_VMAX : FbAnalogValue_Medium (2116) := (                _sDescription := 'Største luftmengde',                 _rCov_Increment := 1,                 _eUnits := WagoTypesBacnet.eBACnetUnits.UNIT_CUBIC_METERS_PER_HOUR           );
  A_360_01_SQ4_A401_0_FB : FbAnalogInput_Medium (2077) := (                _sDescription := 'Spjeldvinkel',                 _rCov_Increment := 1,                 _eUnits := WagoTypesBacnet.eBACnetUnits.UNIT_PERCENT           );
  A_360_01_SQ4_A401_0_C : FbAnalogOutput_Medium (2038) := (                _sDescription := 'Pådrag',                 _rCov_Increment := 1,                 _eUnits := WagoTypesBacnet.eBACnetUnits.UNIT_PERCENT           );
  A_360_01_SQ4_A401_0_KMD : FbMultiStateValue_Large (2038) := (                _sDescription := 'Manuell overstyring',                 _udiNumberOfStates := 8           );
  A_360_01_SQ4_A401_0_OPT_EKSKL : FbBinaryValue_Medium (2038) := (                _sDescription := 'Optimizer',                 _sActiveText := 'Utkoblet',                 _sInactiveText := 'Innkoblet'           );
  A_360_01_SQ4_A401_0_A1 : FbBinaryInput_Large (2076) := (                _sDescription := 'Luftmengde Sjeld',                 _sActiveText := 'Feil på luftmengde',                 _sInactiveText := 'Ingen feil',                 _udiNotificationClass := 22           );
  A_360_01_SQ4_A401_0_A2 : FbBinaryInput_Large (2077) := (                _sDescription := 'Kommunikasjonovervåking',                 _sActiveText := 'Kommunikasjonsfeil',                 _sInactiveText := 'Ingen feil',                 _udiNotificationClass := 22           );
  A_360_01_SQ4_A426_VOL : FbAnalogInput_Medium (2078) := (                _sDescription := 'Faktisk luftmengde',                 _rCov_Increment := 1,                 _eUnits := WagoTypesBacnet.eBACnetUnits.UNIT_CUBIC_METERS_PER_HOUR           );
  A_360_01_SQ4_A426_SP : FbAnalogValue_Medium (2117) := (                _sDescription := 'Settpunkt',                 _rCov_Increment := 1,                 _eUnits := WagoTypesBacnet.eBACnetUnits.UNIT_CUBIC_METERS_PER_HOUR           );
  A_360_01_SQ4_A426_VMIN : FbAnalogValue_Medium (2118) := (                _sDescription := 'Minste luftmengde',                 _rCov_Increment := 1,                 _eUnits := WagoTypesBacnet.eBACnetUnits.UNIT_CUBIC_METERS_PER_HOUR           );
  A_360_01_SQ4_A426_VMAX : FbAnalogValue_Medium (2119) := (                _sDescription := 'Største luftmengde',                 _rCov_Increment := 1,                 _eUnits := WagoTypesBacnet.eBACnetUnits.UNIT_CUBIC_METERS_PER_HOUR           );
  A_360_01_SQ4_A426_FB : FbAnalogInput_Medium (2079) := (                _sDescription := 'Spjeldvinkel',                 _rCov_Increment := 1,                 _eUnits := WagoTypesBacnet.eBACnetUnits.UNIT_PERCENT           );
  A_360_01_SQ4_A426_C : FbAnalogOutput_Medium (2039) := (                _sDescription := 'Pådrag',                 _rCov_Increment := 1,                 _eUnits := WagoTypesBacnet.eBACnetUnits.UNIT_PERCENT           );
  A_360_01_SQ4_A426_KMD : FbMultiStateValue_Large (2039) := (                _sDescription := 'Manuell overstyring',                 _udiNumberOfStates := 8           );
  A_360_01_SQ4_A426_OPT_EKSKL : FbBinaryValue_Medium (2039) := (                _sDescription := 'Optimizer',                 _sActiveText := 'Utkoblet',                 _sInactiveText := 'Innkoblet'           );
  A_360_01_SQ4_A426_A1 : FbBinaryInput_Large (2078) := (                _sDescription := 'Luftmengde Sjeld',                 _sActiveText := 'Feil på luftmengde',                 _sInactiveText := 'Ingen feil',                 _udiNotificationClass := 22           );
  A_360_01_SQ4_A426_A2 : FbBinaryInput_Large (2079) := (                _sDescription := 'Kommunikasjonovervåking',                 _sActiveText := 'Kommunikasjonsfeil',                 _sInactiveText := 'Ingen feil',                 _udiNotificationClass := 22           );
  A_360_01_SQ4_A428_1_VOL : FbAnalogInput_Medium (2080) := (                _sDescription := 'Faktisk luftmengde',                 _rCov_Increment := 1,                 _eUnits := WagoTypesBacnet.eBACnetUnits.UNIT_CUBIC_METERS_PER_HOUR           );
  A_360_01_SQ4_A428_1_SP : FbAnalogValue_Medium (2120) := (                _sDescription := 'Settpunkt',                 _rCov_Increment := 1,                 _eUnits := WagoTypesBacnet.eBACnetUnits.UNIT_CUBIC_METERS_PER_HOUR           );
  A_360_01_SQ4_A428_1_VMIN : FbAnalogValue_Medium (2121) := (                _sDescription := 'Minste luftmengde',                 _rCov_Increment := 1,                 _eUnits := WagoTypesBacnet.eBACnetUnits.UNIT_CUBIC_METERS_PER_HOUR           );
  A_360_01_SQ4_A428_1_VMAX : FbAnalogValue_Medium (2122) := (                _sDescription := 'Største luftmengde',                 _rCov_Increment := 1,                 _eUnits := WagoTypesBacnet.eBACnetUnits.UNIT_CUBIC_METERS_PER_HOUR           );
  A_360_01_SQ4_A428_1_FB : FbAnalogInput_Medium (2081) := (                _sDescription := 'Spjeldvinkel',                 _rCov_Increment := 1,                 _eUnits := WagoTypesBacnet.eBACnetUnits.UNIT_PERCENT           );
  A_360_01_SQ4_A428_1_C : FbAnalogOutput_Medium (2040) := (                _sDescription := 'Pådrag',                 _rCov_Increment := 1,                 _eUnits := WagoTypesBacnet.eBACnetUnits.UNIT_PERCENT           );
  A_360_01_SQ4_A428_1_KMD : FbMultiStateValue_Large (2040) := (                _sDescription := 'Manuell overstyring',                 _udiNumberOfStates := 8           );
  A_360_01_SQ4_A428_1_OPT_EKSKL : FbBinaryValue_Medium (2040) := (                _sDescription := 'Optimizer',                 _sActiveText := 'Utkoblet',                 _sInactiveText := 'Innkoblet'           );
  A_360_01_SQ4_A428_1_A1 : FbBinaryInput_Large (2080) := (                _sDescription := 'Luftmengde Sjeld',                 _sActiveText := 'Feil på luftmengde',                 _sInactiveText := 'Ingen feil',                 _udiNotificationClass := 22           );
  A_360_01_SQ4_A428_1_A2 : FbBinaryInput_Large (2081) := (                _sDescription := 'Kommunikasjonovervåking',                 _sActiveText := 'Kommunikasjonsfeil',                 _sInactiveText := 'Ingen feil',                 _udiNotificationClass := 22           );
  A_360_01_SQ4_A428_2_VOL : FbAnalogInput_Medium (2082) := (                _sDescription := 'Faktisk luftmengde',                 _rCov_Increment := 1,                 _eUnits := WagoTypesBacnet.eBACnetUnits.UNIT_CUBIC_METERS_PER_HOUR           );
  A_360_01_SQ4_A428_2_SP : FbAnalogValue_Medium (2123) := (                _sDescription := 'Settpunkt',                 _rCov_Increment := 1,                 _eUnits := WagoTypesBacnet.eBACnetUnits.UNIT_CUBIC_METERS_PER_HOUR           );
  A_360_01_SQ4_A428_2_VMIN : FbAnalogValue_Medium (2124) := (                _sDescription := 'Minste luftmengde',                 _rCov_Increment := 1,                 _eUnits := WagoTypesBacnet.eBACnetUnits.UNIT_CUBIC_METERS_PER_HOUR           );
  A_360_01_SQ4_A428_2_VMAX : FbAnalogValue_Medium (2125) := (                _sDescription := 'Største luftmengde',                 _rCov_Increment := 1,                 _eUnits := WagoTypesBacnet.eBACnetUnits.UNIT_CUBIC_METERS_PER_HOUR           );
  A_360_01_SQ4_A428_2_FB : FbAnalogInput_Medium (2083) := (                _sDescription := 'Spjeldvinkel',                 _rCov_Increment := 1,                 _eUnits := WagoTypesBacnet.eBACnetUnits.UNIT_PERCENT           );
  A_360_01_SQ4_A428_2_C : FbAnalogOutput_Medium (2041) := (                _sDescription := 'Pådrag',                 _rCov_Increment := 1,                 _eUnits := WagoTypesBacnet.eBACnetUnits.UNIT_PERCENT           );
  A_360_01_SQ4_A428_2_KMD : FbMultiStateValue_Large (2041) := (                _sDescription := 'Manuell overstyring',                 _udiNumberOfStates := 8           );
  A_360_01_SQ4_A428_2_OPT_EKSKL : FbBinaryValue_Medium (2041) := (                _sDescription := 'Optimizer',                 _sActiveText := 'Utkoblet',                 _sInactiveText := 'Innkoblet'           );
  A_360_01_SQ4_A428_2_A1 : FbBinaryInput_Large (2082) := (                _sDescription := 'Luftmengde Sjeld',                 _sActiveText := 'Feil på luftmengde',                 _sInactiveText := 'Ingen feil',                 _udiNotificationClass := 22           );
  A_360_01_SQ4_A428_2_A2 : FbBinaryInput_Large (2083) := (                _sDescription := 'Kommunikasjonovervåking',                 _sActiveText := 'Kommunikasjonsfeil',                 _sInactiveText := 'Ingen feil',                 _udiNotificationClass := 22           );
  A_360_01_SQ4_A428_3_VOL : FbAnalogInput_Medium (2084) := (                _sDescription := 'Faktisk luftmengde',                 _rCov_Increment := 1,                 _eUnits := WagoTypesBacnet.eBACnetUnits.UNIT_CUBIC_METERS_PER_HOUR           );
  A_360_01_SQ4_A428_3_SP : FbAnalogValue_Medium (2126) := (                _sDescription := 'Settpunkt',                 _rCov_Increment := 1,                 _eUnits := WagoTypesBacnet.eBACnetUnits.UNIT_CUBIC_METERS_PER_HOUR           );
  A_360_01_SQ4_A428_3_VMIN : FbAnalogValue_Medium (2127) := (                _sDescription := 'Minste luftmengde',                 _rCov_Increment := 1,                 _eUnits := WagoTypesBacnet.eBACnetUnits.UNIT_CUBIC_METERS_PER_HOUR           );
  A_360_01_SQ4_A428_3_VMAX : FbAnalogValue_Medium (2128) := (                _sDescription := 'Største luftmengde',                 _rCov_Increment := 1,                 _eUnits := WagoTypesBacnet.eBACnetUnits.UNIT_CUBIC_METERS_PER_HOUR           );
  A_360_01_SQ4_A428_3_FB : FbAnalogInput_Medium (2085) := (                _sDescription := 'Spjeldvinkel',                 _rCov_Increment := 1,                 _eUnits := WagoTypesBacnet.eBACnetUnits.UNIT_PERCENT           );
  A_360_01_SQ4_A428_3_C : FbAnalogOutput_Medium (2042) := (                _sDescription := 'Pådrag',                 _rCov_Increment := 1,                 _eUnits := WagoTypesBacnet.eBACnetUnits.UNIT_PERCENT           );
  A_360_01_SQ4_A428_3_KMD : FbMultiStateValue_Large (2042) := (                _sDescription := 'Manuell overstyring',                 _udiNumberOfStates := 8           );
  A_360_01_SQ4_A428_3_OPT_EKSKL : FbBinaryValue_Medium (2042) := (                _sDescription := 'Optimizer',                 _sActiveText := 'Utkoblet',                 _sInactiveText := 'Innkoblet'           );
  A_360_01_SQ4_A428_3_A1 : FbBinaryInput_Large (2084) := (                _sDescription := 'Luftmengde Sjeld',                 _sActiveText := 'Feil på luftmengde',                 _sInactiveText := 'Ingen feil',                 _udiNotificationClass := 22           );
  A_360_01_SQ4_A428_3_A2 : FbBinaryInput_Large (2085) := (                _sDescription := 'Kommunikasjonovervåking',                 _sActiveText := 'Kommunikasjonsfeil',                 _sInactiveText := 'Ingen feil',                 _udiNotificationClass := 22           );
  A_360_01_SQ4_A428_4_VOL : FbAnalogInput_Medium (2086) := (                _sDescription := 'Faktisk luftmengde',                 _rCov_Increment := 1,                 _eUnits := WagoTypesBacnet.eBACnetUnits.UNIT_CUBIC_METERS_PER_HOUR           );
  A_360_01_SQ4_A428_4_SP : FbAnalogValue_Medium (2129) := (                _sDescription := 'Settpunkt',                 _rCov_Increment := 1,                 _eUnits := WagoTypesBacnet.eBACnetUnits.UNIT_CUBIC_METERS_PER_HOUR           );
  A_360_01_SQ4_A428_4_VMIN : FbAnalogValue_Medium (2130) := (                _sDescription := 'Minste luftmengde',                 _rCov_Increment := 1,                 _eUnits := WagoTypesBacnet.eBACnetUnits.UNIT_CUBIC_METERS_PER_HOUR           );
  A_360_01_SQ4_A428_4_VMAX : FbAnalogValue_Medium (2131) := (                _sDescription := 'Største luftmengde',                 _rCov_Increment := 1,                 _eUnits := WagoTypesBacnet.eBACnetUnits.UNIT_CUBIC_METERS_PER_HOUR           );
  A_360_01_SQ4_A428_4_FB : FbAnalogInput_Medium (2087) := (                _sDescription := 'Spjeldvinkel',                 _rCov_Increment := 1,                 _eUnits := WagoTypesBacnet.eBACnetUnits.UNIT_PERCENT           );
  A_360_01_SQ4_A428_4_C : FbAnalogOutput_Medium (2043) := (                _sDescription := 'Pådrag',                 _rCov_Increment := 1,                 _eUnits := WagoTypesBacnet.eBACnetUnits.UNIT_PERCENT           );
  A_360_01_SQ4_A428_4_KMD : FbMultiStateValue_Large (2043) := (                _sDescription := 'Manuell overstyring',                 _udiNumberOfStates := 8           );
  A_360_01_SQ4_A428_4_OPT_EKSKL : FbBinaryValue_Medium (2043) := (                _sDescription := 'Optimizer',                 _sActiveText := 'Utkoblet',                 _sInactiveText := 'Innkoblet'           );
  A_360_01_SQ4_A428_4_A1 : FbBinaryInput_Large (2086) := (                _sDescription := 'Luftmengde Sjeld',                 _sActiveText := 'Feil på luftmengde',                 _sInactiveText := 'Ingen feil',                 _udiNotificationClass := 22           );
  A_360_01_SQ4_A428_4_A2 : FbBinaryInput_Large (2087) := (                _sDescription := 'Kommunikasjonovervåking',                 _sActiveText := 'Kommunikasjonsfeil',                 _sInactiveText := 'Ingen feil',                 _udiNotificationClass := 22           );
  A_360_01_SQ5_A425_VOL : FbAnalogInput_Medium (2088) := (                _sDescription := 'Faktisk luftmengde',                 _rCov_Increment := 1,                 _eUnits := WagoTypesBacnet.eBACnetUnits.UNIT_CUBIC_METERS_PER_HOUR           );
  A_360_01_SQ5_A425_SP : FbAnalogValue_Medium (2132) := (                _sDescription := 'Settpunkt',                 _rCov_Increment := 1,                 _eUnits := WagoTypesBacnet.eBACnetUnits.UNIT_CUBIC_METERS_PER_HOUR           );
  A_360_01_SQ5_A425_VMIN : FbAnalogValue_Medium (2133) := (                _sDescription := 'Minste luftmengde',                 _rCov_Increment := 1,                 _eUnits := WagoTypesBacnet.eBACnetUnits.UNIT_CUBIC_METERS_PER_HOUR           );
  A_360_01_SQ5_A425_VMAX : FbAnalogValue_Medium (2134) := (                _sDescription := 'Største luftmengde',                 _rCov_Increment := 1,                 _eUnits := WagoTypesBacnet.eBACnetUnits.UNIT_CUBIC_METERS_PER_HOUR           );
  A_360_01_SQ5_A425_FB : FbAnalogInput_Medium (2089) := (                _sDescription := 'Spjeldvinkel',                 _rCov_Increment := 1,                 _eUnits := WagoTypesBacnet.eBACnetUnits.UNIT_PERCENT           );
  A_360_01_SQ5_A425_C : FbAnalogOutput_Medium (2044) := (                _sDescription := 'Pådrag',                 _rCov_Increment := 1,                 _eUnits := WagoTypesBacnet.eBACnetUnits.UNIT_PERCENT           );
  A_360_01_SQ5_A425_KMD : FbMultiStateValue_Large (2044) := (                _sDescription := 'Manuell overstyring',                 _udiNumberOfStates := 8           );
  A_360_01_SQ5_A425_OPT_EKSKL : FbBinaryValue_Medium (2044) := (                _sDescription := 'Optimizer',                 _sActiveText := 'Utkoblet',                 _sInactiveText := 'Innkoblet'           );
  A_360_01_SQ5_A425_A1 : FbBinaryInput_Large (2088) := (                _sDescription := 'Luftmengde Sjeld',                 _sActiveText := 'Feil på luftmengde',                 _sInactiveText := 'Ingen feil',                 _udiNotificationClass := 22           );
  A_360_01_SQ5_A425_A2 : FbBinaryInput_Large (2089) := (                _sDescription := 'Kommunikasjonovervåking',                 _sActiveText := 'Kommunikasjonsfeil',                 _sInactiveText := 'Ingen feil',                 _udiNotificationClass := 22           );
  A_360_01_SQ4_A428_5_VOL : FbAnalogInput_Medium (2090) := (                _sDescription := 'Faktisk luftmengde',                 _rCov_Increment := 1,                 _eUnits := WagoTypesBacnet.eBACnetUnits.UNIT_CUBIC_METERS_PER_HOUR           );
  A_360_01_SQ4_A428_5_SP : FbAnalogValue_Medium (2135) := (                _sDescription := 'Settpunkt',                 _rCov_Increment := 1,                 _eUnits := WagoTypesBacnet.eBACnetUnits.UNIT_CUBIC_METERS_PER_HOUR           );
  A_360_01_SQ4_A428_5_VMIN : FbAnalogValue_Medium (2136) := (                _sDescription := 'Minste luftmengde',                 _rCov_Increment := 1,                 _eUnits := WagoTypesBacnet.eBACnetUnits.UNIT_CUBIC_METERS_PER_HOUR           );
  A_360_01_SQ4_A428_5_VMAX : FbAnalogValue_Medium (2137) := (                _sDescription := 'Største luftmengde',                 _rCov_Increment := 1,                 _eUnits := WagoTypesBacnet.eBACnetUnits.UNIT_CUBIC_METERS_PER_HOUR           );
  A_360_01_SQ4_A428_5_FB : FbAnalogInput_Medium (2091) := (                _sDescription := 'Spjeldvinkel',                 _rCov_Increment := 1,                 _eUnits := WagoTypesBacnet.eBACnetUnits.UNIT_PERCENT           );
  A_360_01_SQ4_A428_5_C : FbAnalogOutput_Medium (2045) := (                _sDescription := 'Pådrag',                 _rCov_Increment := 1,                 _eUnits := WagoTypesBacnet.eBACnetUnits.UNIT_PERCENT           );
  A_360_01_SQ4_A428_5_KMD : FbMultiStateValue_Large (2045) := (                _sDescription := 'Manuell overstyring',                 _udiNumberOfStates := 8           );
  A_360_01_SQ4_A428_5_OPT_EKSKL : FbBinaryValue_Medium (2045) := (                _sDescription := 'Optimizer',                 _sActiveText := 'Utkoblet',                 _sInactiveText := 'Innkoblet'           );
  A_360_01_SQ4_A428_5_A1 : FbBinaryInput_Large (2090) := (                _sDescription := 'Luftmengde Sjeld',                 _sActiveText := 'Feil på luftmengde',                 _sInactiveText := 'Ingen feil',                 _udiNotificationClass := 22           );
  A_360_01_SQ4_A428_5_A2 : FbBinaryInput_Large (2091) := (                _sDescription := 'Kommunikasjonovervåking',                 _sActiveText := 'Kommunikasjonsfeil',                 _sInactiveText := 'Ingen feil',                 _udiNotificationClass := 22           );
  A_360_01_SQ4_A428_6_VOL : FbAnalogInput_Medium (2092) := (                _sDescription := 'Faktisk luftmengde',                 _rCov_Increment := 1,                 _eUnits := WagoTypesBacnet.eBACnetUnits.UNIT_CUBIC_METERS_PER_HOUR           );
  A_360_01_SQ4_A428_6_SP : FbAnalogValue_Medium (2138) := (                _sDescription := 'Settpunkt',                 _rCov_Increment := 1,                 _eUnits := WagoTypesBacnet.eBACnetUnits.UNIT_CUBIC_METERS_PER_HOUR           );
  A_360_01_SQ4_A428_6_VMIN : FbAnalogValue_Medium (2139) := (                _sDescription := 'Minste luftmengde',                 _rCov_Increment := 1,                 _eUnits := WagoTypesBacnet.eBACnetUnits.UNIT_CUBIC_METERS_PER_HOUR           );
  A_360_01_SQ4_A428_6_VMAX : FbAnalogValue_Medium (2140) := (                _sDescription := 'Største luftmengde',                 _rCov_Increment := 1,                 _eUnits := WagoTypesBacnet.eBACnetUnits.UNIT_CUBIC_METERS_PER_HOUR           );
  A_360_01_SQ4_A428_6_FB : FbAnalogInput_Medium (2093) := (                _sDescription := 'Spjeldvinkel',                 _rCov_Increment := 1,                 _eUnits := WagoTypesBacnet.eBACnetUnits.UNIT_PERCENT           );
  A_360_01_SQ4_A428_6_C : FbAnalogOutput_Medium (2046) := (                _sDescription := 'Pådrag',                 _rCov_Increment := 1,                 _eUnits := WagoTypesBacnet.eBACnetUnits.UNIT_PERCENT           );
  A_360_01_SQ4_A428_6_KMD : FbMultiStateValue_Large (2046) := (                _sDescription := 'Manuell overstyring',                 _udiNumberOfStates := 8           );
  A_360_01_SQ4_A428_6_OPT_EKSKL : FbBinaryValue_Medium (2046) := (                _sDescription := 'Optimizer',                 _sActiveText := 'Utkoblet',                 _sInactiveText := 'Innkoblet'           );
  A_360_01_SQ4_A428_6_A1 : FbBinaryInput_Large (2092) := (                _sDescription := 'Luftmengde Sjeld',                 _sActiveText := 'Feil på luftmengde',                 _sInactiveText := 'Ingen feil',                 _udiNotificationClass := 22           );
  A_360_01_SQ4_A428_6_A2 : FbBinaryInput_Large (2093) := (                _sDescription := 'Kommunikasjonovervåking',                 _sActiveText := 'Kommunikasjonsfeil',                 _sInactiveText := 'Ingen feil',                 _udiNotificationClass := 22           );
